LIN {X 0,Y 190.202,Z 1213.13,A -85,B 0,C 180,E1 7235.052,E2 7235.052} C_VEL
LIN {X 0,Y 181.656,Z 1215.666,A -85,B 0,C 180,E1 7232.27,E2 7232.27} C_VEL
LIN {X 0,Y 170.699,Z 1218.765,A -85,B 0,C 180,E1 7227.565,E2 7227.565} C_VEL
LIN {X 0,Y 162.904,Z 1221.055,A -85,B 0,C 180,E1 7223.131,E2 7223.131} C_VEL
LIN {X 0,Y 156.495,Z 1223.066,A -85,B 0,C 180,E1 7218.245,E2 7218.245} C_VEL
LIN {X 0,Y 151.281,Z 1224.964,A -85,B 0,C 180,E1 7212.599,E2 7212.599} C_VEL
LIN {X 0,Y 147.668,Z 1226.836,A -85,B 0,C 180,E1 7206.611,E2 7206.611} C_VEL
LIN {X 0,Y 145.616,Z 1229.303,A -85,B 0,C 180,E1 7198.033,E2 7198.033} C_VEL
LIN {X 0,Y 147.248,Z 1232.369,A -85,B 0,C 180,E1 7187.849,E2 7187.849} C_VEL
LIN {X 0,Y 157.913,Z 1236.155,A -85,B 0,C 180,E1 7174.498,E2 7174.498} C_VEL
LIN {X 0,Y 172.688,Z 1238.099,A -85,B 0,C 180,E1 7165.832,E2 7165.832} C_VEL
LIN {X 0,Y 175.368,Z 1238.372,A -85,B 0,C 180,E1 7164.62,E2 7164.62} C_VEL
LIN {X 0,Y 164.681,Z 1250.11,A -85,B 0,C 180,E1 7159.372,E2 7159.372} C_VEL
LIN {X 0,Y 155.017,Z 1260.363,A -85,B 0,C 180,E1 7153.135,E2 7153.135} C_VEL
LIN {X 0,Y 147.162,Z 1268.783,A -85,B 0,C 180,E1 7146.123,E2 7146.123} C_VEL
LIN {X 0,Y 143.911,Z 1271.432,A -85,B 0,C 180,E1 7143.535,E2 7143.535} C_VEL
LIN {X 0,Y 132.963,Z 1277.212,A -85,B 0,C 180,E1 7136.373,E2 7136.373} C_VEL
LIN {X 0,Y 131.052,Z 1278.703,A -85,B 0,C 180,E1 7133.675,E2 7133.675} C_VEL
LIN {X 0,Y 128.932,Z 1282.473,A -85,B 0,C 180,E1 7124.83,E2 7124.83} C_VEL
LIN {X 0,Y 128.699,Z 1284.323,A -85,B 0,C 180,E1 7117.143,E2 7117.143} C_VEL
LIN {X 0,Y 128.951,Z 1284.94,A -85,B 0,C 180,E1 7110.891,E2 7110.891} C_VEL
LIN {X 0,Y 128.784,Z 1284.684,A -85,B 0,C 180,E1 7105.103,E2 7105.103} C_VEL
LIN {X 0,Y 128.69,Z 1283.094,A -85,B 0,C 180,E1 7097.437,E2 7097.437} C_VEL
LIN {X 0,Y 130.24,Z 1279.703,A -85,B 0,C 180,E1 7088.379,E2 7088.379} C_VEL
LIN {X 0,Y 134.227,Z 1274.587,A -85,B 0,C 180,E1 7079.569,E2 7079.569} C_VEL
LIN {X 0,Y 141.174,Z 1267.225,A -85,B 0,C 180,E1 7070.927,E2 7070.927} C_VEL
LIN {X 0,Y 150.261,Z 1258.18,A -85,B 0,C 180,E1 7063.509,E2 7063.509} C_VEL
LIN {X 0,Y 160.858,Z 1247.554,A -85,B 0,C 180,E1 7057.289,E2 7057.289} C_VEL
LIN {X 0,Y 171.789,Z 1236.049,A -85,B 0,C 180,E1 7052.375,E2 7052.375} C_VEL
LIN {X 0,Y 183.624,Z 1222.614,A -85,B 0,C 180,E1 7048.105,E2 7048.105} C_VEL
LIN {X 0,Y 195.661,Z 1207.553,A -85,B 0,C 180,E1 7044.553,E2 7044.553} C_VEL
LIN {X 0,Y 206.741,Z 1192.05,A -85,B 0,C 180,E1 7041.792,E2 7041.792} C_VEL
LIN {X 0,Y 217.435,Z 1175.098,A -85,B 0,C 180,E1 7039.498,E2 7039.498} C_VEL
LIN {X 0,Y 227.58,Z 1156.363,A -85,B 0,C 180,E1 7037.57,E2 7037.57} C_VEL
LIN {X 0,Y 236.655,Z 1136.35,A -85,B 0,C 180,E1 7036.022,E2 7036.022} C_VEL
LIN {X 0,Y 244.117,Z 1116.061,A -85,B 0,C 180,E1 7034.852,E2 7034.852} C_VEL
LIN {X 0,Y 249.756,Z 1096.487,A -85,B 0,C 180,E1 7034.032,E2 7034.032} C_VEL
LIN {X 0,Y 254.152,Z 1075.647,A -85,B 0,C 180,E1 7033.393,E2 7033.393} C_VEL
LIN {X 0,Y 257.474,Z 1050.007,A -85,B 0,C 180,E1 7032.818,E2 7032.818} C_VEL
LIN {X 0,Y 260.557,Z 1021.82,A -85,B 0,C 180,E1 7032.373,E2 7032.373} C_VEL
LIN {X 0,Y 264.495,Z 989.715,A -85,B 0,C 180,E1 7032.277,E2 7032.277} C_VEL
LIN {X 0,Y 264.76,Z 957.802,A -85,B 0,C 180,E1 7027.95,E2 7027.95} C_VEL
LIN {X 0,Y 266.442,Z 929.886,A -85,B 0,C 180,E1 7024.735,E2 7024.735} C_VEL
LIN {X 0,Y 266.944,Z 923.717,A -85,B 0,C 180,E1 7024.08,E2 7024.08} C_VEL
LIN {X 0,Y 267.411,Z 913.202,A -85,B 0,C 180,E1 7019.41,E2 7019.41} C_VEL
LIN {X 0,Y 268.624,Z 906.957,A -85,B 0,C 180,E1 7016.265,E2 7016.265} C_VEL
LIN {X 0,Y 271.7,Z 898.866,A -85,B 0,C 180,E1 7011.748,E2 7011.748} C_VEL
LIN {X 0,Y 277.101,Z 891.459,A -85,B 0,C 180,E1 7006.648,E2 7006.648} C_VEL
LIN {X 0,Y 277.44,Z 891.39,A -85,B 0,C 180,E1 7006.354,E2 7006.354} C_VEL
LIN {X 0,Y 259.966,Z 1057.824,A -85,B 0,C 180,E1 7003.172,E2 7003.172} C_VEL
LIN {X 0,Y 256.354,Z 1078.331,A -85,B 0,C 180,E1 7002.543,E2 7002.543} C_VEL
LIN {X 0,Y 251.132,Z 1098.893,A -85,B 0,C 180,E1 7001.667,E2 7001.667} C_VEL
LIN {X 0,Y 244.438,Z 1118.855,A -85,B 0,C 180,E1 7000.531,E2 7000.531} C_VEL
LIN {X 0,Y 236.901,Z 1136.955,A -85,B 0,C 180,E1 6999.202,E2 6999.202} C_VEL
LIN {X 0,Y 228.237,Z 1154.356,A -85,B 0,C 180,E1 6997.566,E2 6997.566} C_VEL
LIN {X 0,Y 218.015,Z 1171.667,A -85,B 0,C 180,E1 6995.468,E2 6995.468} C_VEL
LIN {X 0,Y 207.123,Z 1187.56,A -85,B 0,C 180,E1 6992.952,E2 6992.952} C_VEL
LIN {X 0,Y 195.887,Z 1201.926,A -85,B 0,C 180,E1 6989.985,E2 6989.985} C_VEL
LIN {X 0,Y 183.923,Z 1215.491,A -85,B 0,C 180,E1 6986.276,E2 6986.276} C_VEL
LIN {X 0,Y 171.894,Z 1227.707,A -85,B 0,C 180,E1 6981.741,E2 6981.741} C_VEL
LIN {X 0,Y 160.986,Z 1237.804,A -85,B 0,C 180,E1 6976.605,E2 6976.605} C_VEL
LIN {X 0,Y 150.926,Z 1246.477,A -85,B 0,C 180,E1 6970.481,E2 6970.481} C_VEL
LIN {X 0,Y 142.092,Z 1253.744,A -85,B 0,C 180,E1 6963.135,E2 6963.135} C_VEL
LIN {X 0,Y 135.409,Z 1259.191,A -85,B 0,C 180,E1 6954.888,E2 6954.888} C_VEL
LIN {X 0,Y 131.267,Z 1262.741,A -85,B 0,C 180,E1 6946.31,E2 6946.31} C_VEL
LIN {X 0,Y 129.3,Z 1264.71,A -85,B 0,C 180,E1 6937.552,E2 6937.552} C_VEL
LIN {X 0,Y 128.89,Z 1265.289,A -85,B 0,C 180,E1 6929.554,E2 6929.554} C_VEL
LIN {X 0,Y 129.406,Z 1264.614,A -85,B 0,C 180,E1 6921.556,E2 6921.556} C_VEL
LIN {X 0,Y 131.568,Z 1262.487,A -85,B 0,C 180,E1 6912.758,E2 6912.758} C_VEL
LIN {X 0,Y 135.899,Z 1258.805,A -85,B 0,C 180,E1 6904.271,E2 6904.271} C_VEL
LIN {X 0,Y 142.537,Z 1253.449,A -85,B 0,C 180,E1 6896.345,E2 6896.345} C_VEL
LIN {X 0,Y 151.344,Z 1246.237,A -85,B 0,C 180,E1 6889.151,E2 6889.151} C_VEL
LIN {X 0,Y 161.477,Z 1237.497,A -85,B 0,C 180,E1 6883.057,E2 6883.057} C_VEL
LIN {X 0,Y 172.614,Z 1227.163,A -85,B 0,C 180,E1 6877.88,E2 6877.88} C_VEL
LIN {X 0,Y 180.192,Z 1219.524,A -85,B 0,C 180,E1 6874.858,E2 6874.858} C_VEL
LIN {X 0,Y 166.021,Z 1223.23,A -85,B 0,C 180,E1 6869.198,E2 6869.198} C_VEL
LIN {X 0,Y 157.334,Z 1225.582,A -85,B 0,C 180,E1 6864.399,E2 6864.399} C_VEL
LIN {X 0,Y 150.611,Z 1227.559,A -85,B 0,C 180,E1 6859.387,E2 6859.387} C_VEL
LIN {X 0,Y 145.112,Z 1229.463,A -85,B 0,C 180,E1 6853.549,E2 6853.549} C_VEL
LIN {X 0,Y 141.144,Z 1231.414,A -85,B 0,C 180,E1 6846.918,E2 6846.918} C_VEL
LIN {X 0,Y 139.007,Z 1233.771,A -85,B 0,C 180,E1 6838.352,E2 6838.352} C_VEL
LIN {X 0,Y 140.751,Z 1236.859,A -85,B 0,C 180,E1 6827.279,E2 6827.279} C_VEL
LIN {X 0,Y 151.475,Z 1240.492,A -85,B 0,C 180,E1 6813.753,E2 6813.753} C_VEL
LIN {X 0,Y 166.114,Z 1242.561,A -85,B 0,C 180,E1 6804.947,E2 6804.947} C_VEL
LIN {X 0,Y 155.353,Z 1253.519,A -85,B 0,C 180,E1 6799.418,E2 6799.418} C_VEL
LIN {X 0,Y 145.567,Z 1263.173,A -85,B 0,C 180,E1 6792.698,E2 6792.698} C_VEL
LIN {X 0,Y 137.392,Z 1271.411,A -85,B 0,C 180,E1 6784.588,E2 6784.588} C_VEL
LIN {X 0,Y 131.799,Z 1277.771,A -85,B 0,C 180,E1 6775.478,E2 6775.478} C_VEL
LIN {X 0,Y 131.052,Z 1278.703,A -85,B 0,C 180,E1 6773.675,E2 6773.675} C_VEL
LIN {X 0,Y 129.012,Z 1280.314,A -85,B 0,C 180,E1 6770.444,E2 6770.444} C_VEL
LIN {X 0,Y 123.443,Z 1282.376,A -85,B 0,C 180,E1 6764.399,E2 6764.399} C_VEL
LIN {X 0,Y 120.803,Z 1283.402,A -85,B 0,C 180,E1 6759.575,E2 6759.575} C_VEL
LIN {X 0,Y 120.68,Z 1283.603,A -85,B 0,C 180,E1 6758.252,E2 6758.252} C_VEL
LIN {X 0,Y 120.946,Z 1284.28,A -85,B 0,C 180,E1 6751.897,E2 6751.897} C_VEL
LIN {X 0,Y 120.862,Z 1284.165,A -85,B 0,C 180,E1 6746.207,E2 6746.207} C_VEL
LIN {X 0,Y 120.653,Z 1282.984,A -85,B 0,C 180,E1 6738.53,E2 6738.53} C_VEL
LIN {X 0,Y 121.897,Z 1280.096,A -85,B 0,C 180,E1 6729.349,E2 6729.349} C_VEL
LIN {X 0,Y 125.732,Z 1275.36,A -85,B 0,C 180,E1 6719.937,E2 6719.937} C_VEL
LIN {X 0,Y 132.369,Z 1268.778,A -85,B 0,C 180,E1 6711.078,E2 6711.078} C_VEL
LIN {X 0,Y 141.438,Z 1260.425,A -85,B 0,C 180,E1 6703.273,E2 6703.273} C_VEL
LIN {X 0,Y 151.584,Z 1251.084,A -85,B 0,C 180,E1 6697.052,E2 6697.052} C_VEL
LIN {X 0,Y 163.215,Z 1239.802,A -85,B 0,C 180,E1 6691.627,E2 6691.627} C_VEL
LIN {X 0,Y 176.089,Z 1226.257,A -85,B 0,C 180,E1 6686.945,E2 6686.945} C_VEL
LIN {X 0,Y 188.388,Z 1211.935,A -85,B 0,C 180,E1 6683.342,E2 6683.342} C_VEL
LIN {X 0,Y 199.998,Z 1196.799,A -85,B 0,C 180,E1 6680.484,E2 6680.484} C_VEL
LIN {X 0,Y 211.415,Z 1179.946,A -85,B 0,C 180,E1 6678.089,E2 6678.089} C_VEL
LIN {X 0,Y 221.752,Z 1162.307,A -85,B 0,C 180,E1 6676.184,E2 6676.184} C_VEL
LIN {X 0,Y 230.796,Z 1144.223,A -85,B 0,C 180,E1 6674.688,E2 6674.688} C_VEL
LIN {X 0,Y 238.814,Z 1124.974,A -85,B 0,C 180,E1 6673.476,E2 6673.476} C_VEL
LIN {X 0,Y 245.784,Z 1103.885,A -85,B 0,C 180,E1 6672.498,E2 6672.498} C_VEL
LIN {X 0,Y 250.857,Z 1083.368,A -85,B 0,C 180,E1 6671.837,E2 6671.837} C_VEL
LIN {X 0,Y 254.306,Z 1062.63,A -85,B 0,C 180,E1 6671.335,E2 6671.335} C_VEL
LIN {X 0,Y 258.057,Z 1029.137,A -85,B 0,C 180,E1 6670.725,E2 6670.725} C_VEL
LIN {X 0,Y 261.533,Z 1000.333,A -85,B 0,C 180,E1 6670.585,E2 6670.585} C_VEL
LIN {X 0,Y 262.564,Z 991.884,A -85,B 0,C 180,E1 6670.557,E2 6670.557} C_VEL
LIN {X 0,Y 263.401,Z 960.962,A -85,B 0,C 180,E1 6666.374,E2 6666.374} C_VEL
LIN {X 0,Y 265.477,Z 933.239,A -85,B 0,C 180,E1 6663.184,E2 6663.184} C_VEL
LIN {X 0,Y 265.825,Z 929.431,A -85,B 0,C 180,E1 6662.748,E2 6662.748} C_VEL
LIN {X 0,Y 266.599,Z 920.148,A -85,B 0,C 180,E1 6658.549,E2 6658.549} C_VEL
LIN {X 0,Y 267.913,Z 914.319,A -85,B 0,C 180,E1 6655.612,E2 6655.612} C_VEL
LIN {X 0,Y 271.136,Z 906.412,A -85,B 0,C 180,E1 6651.197,E2 6651.197} C_VEL
LIN {X 0,Y 274.63,Z 901.489,A -85,B 0,C 180,E1 6647.796,E2 6647.796} C_VEL
LIN {X 0,Y 257.755,Z 1058.451,A -85,B 0,C 180,E1 6644.868,E2 6644.868} C_VEL
LIN {X 0,Y 254.091,Z 1078.81,A -85,B 0,C 180,E1 6644.263,E2 6644.263} C_VEL
LIN {X 0,Y 248.777,Z 1099.339,A -85,B 0,C 180,E1 6643.419,E2 6643.419} C_VEL
LIN {X 0,Y 242.324,Z 1118.342,A -85,B 0,C 180,E1 6642.385,E2 6642.385} C_VEL
LIN {X 0,Y 234.585,Z 1136.721,A -85,B 0,C 180,E1 6641.099,E2 6641.099} C_VEL
LIN {X 0,Y 225.303,Z 1154.957,A -85,B 0,C 180,E1 6639.449,E2 6639.449} C_VEL
LIN {X 0,Y 214.745,Z 1172.372,A -85,B 0,C 180,E1 6637.402,E2 6637.402} C_VEL
LIN {X 0,Y 203.594,Z 1188.167,A -85,B 0,C 180,E1 6634.967,E2 6634.967} C_VEL
LIN {X 0,Y 192.257,Z 1202.219,A -85,B 0,C 180,E1 6632.139,E2 6632.139} C_VEL
LIN {X 0,Y 179.753,Z 1215.917,A -85,B 0,C 180,E1 6628.475,E2 6628.475} C_VEL
LIN {X 0,Y 167.682,Z 1227.709,A -85,B 0,C 180,E1 6624.185,E2 6624.185} C_VEL
LIN {X 0,Y 156.15,Z 1237.926,A -85,B 0,C 180,E1 6619.073,E2 6619.073} C_VEL
LIN {X 0,Y 145.392,Z 1246.707,A -85,B 0,C 180,E1 6612.905,E2 6612.905} C_VEL
LIN {X 0,Y 135.524,Z 1254.267,A -85,B 0,C 180,E1 6605.13,E2 6605.13} C_VEL
LIN {X 0,Y 128.135,Z 1259.807,A -85,B 0,C 180,E1 6596.407,E2 6596.407} C_VEL
LIN {X 0,Y 123.524,Z 1263.398,A -85,B 0,C 180,E1 6587.222,E2 6587.222} C_VEL
LIN {X 0,Y 121.375,Z 1265.321,A -85,B 0,C 180,E1 6578.048,E2 6578.048} C_VEL
LIN {X 0,Y 120.913,Z 1265.897,A -85,B 0,C 180,E1 6569.524,E2 6569.524} C_VEL
LIN {X 0,Y 121.428,Z 1265.285,A -85,B 0,C 180,E1 6561.474,E2 6561.474} C_VEL
LIN {X 0,Y 123.734,Z 1263.249,A -85,B 0,C 180,E1 6552.115,E2 6552.115} C_VEL
LIN {X 0,Y 128.379,Z 1259.659,A -85,B 0,C 180,E1 6543.144,E2 6543.144} C_VEL
LIN {X 0,Y 135.879,Z 1254.064,A -85,B 0,C 180,E1 6534.455,E2 6534.455} C_VEL
LIN {X 0,Y 145.32,Z 1246.851,A -85,B 0,C 180,E1 6527.064,E2 6527.064} C_VEL
LIN {X 0,Y 156.068,Z 1238.11,A -85,B 0,C 180,E1 6520.887,E2 6520.887} C_VEL
LIN {X 0,Y 167.599,Z 1227.933,A -85,B 0,C 180,E1 6515.77,E2 6515.77} C_VEL
LIN {X 0,Y 170.462,Z 1225.224,A -85,B 0,C 180,E1 6514.577,E2 6514.577} C_VEL
LIN {X 0,Y 161.394,Z 1227.526,A -85,B 0,C 180,E1 6510.945,E2 6510.945} C_VEL
LIN {X 0,Y 151.744,Z 1229.936,A -85,B 0,C 180,E1 6505.779,E2 6505.779} C_VEL
LIN {X 0,Y 144.303,Z 1231.953,A -85,B 0,C 180,E1 6500.271,E2 6500.271} C_VEL
LIN {X 0,Y 138.839,Z 1233.726,A -85,B 0,C 180,E1 6494.6,E2 6494.6} C_VEL
LIN {X 0,Y 134.442,Z 1235.714,A -85,B 0,C 180,E1 6487.264,E2 6487.264} C_VEL
LIN {X 0,Y 132.226,Z 1237.88,A -85,B 0,C 180,E1 6479.134,E2 6479.134} C_VEL
LIN {X 0,Y 134.348,Z 1241.242,A -85,B 0,C 180,E1 6466.223,E2 6466.223} C_VEL
LIN {X 0,Y 144.965,Z 1244.651,A -85,B 0,C 180,E1 6452.922,E2 6452.922} C_VEL
LIN {X 0,Y 156.864,Z 1246.466,A -85,B 0,C 180,E1 6445.313,E2 6445.313} C_VEL
LIN {X 0,Y 145.451,Z 1257.166,A -85,B 0,C 180,E1 6439.129,E2 6439.129} C_VEL
LIN {X 0,Y 135.469,Z 1266.256,A -85,B 0,C 180,E1 6431.628,E2 6431.628} C_VEL
LIN {X 0,Y 127.915,Z 1273.369,A -85,B 0,C 180,E1 6423.175,E2 6423.175} C_VEL
LIN {X 0,Y 123.054,Z 1278.667,A -85,B 0,C 180,E1 6413.973,E2 6413.973} C_VEL
LIN {X 0,Y 120.89,Z 1282.238,A -85,B 0,C 180,E1 6404.369,E2 6404.369} C_VEL
LIN {X 0,Y 120.68,Z 1283.603,A -85,B 0,C 180,E1 6398.252,E2 6398.252} C_VEL
LIN {X 0,Y 119.983,Z 1284.024,A -85,B 0,C 180,E1 6395.112,E2 6395.112} C_VEL
LIN {X 0,Y 117.334,Z 1284.085,A -85,B 0,C 180,E1 6390.703,E2 6390.703} C_VEL
LIN {X 0,Y 112.819,Z 1283.189,A -85,B 0,C 180,E1 6382.452,E2 6382.452} C_VEL
LIN {X 0,Y 112.656,Z 1282.948,A -85,B 0,C 180,E1 6381.003,E2 6381.003} C_VEL
LIN {X 0,Y 113.382,Z 1280.71,A -85,B 0,C 180,E1 6371.493,E2 6371.493} C_VEL
LIN {X 0,Y 116.735,Z 1276.632,A -85,B 0,C 180,E1 6361.34,E2 6361.34} C_VEL
LIN {X 0,Y 123.038,Z 1270.723,A -85,B 0,C 180,E1 6351.861,E2 6351.861} C_VEL
LIN {X 0,Y 131.738,Z 1263.271,A -85,B 0,C 180,E1 6343.682,E2 6343.682} C_VEL
LIN {X 0,Y 142.904,Z 1253.731,A -85,B 0,C 180,E1 6336.429,E2 6336.429} C_VEL
LIN {X 0,Y 155.441,Z 1242.448,A -85,B 0,C 180,E1 6330.468,E2 6330.468} C_VEL
LIN {X 0,Y 167.861,Z 1230.368,A -85,B 0,C 180,E1 6325.921,E2 6325.921} C_VEL
LIN {X 0,Y 180.393,Z 1216.979,A -85,B 0,C 180,E1 6322.242,E2 6322.242} C_VEL
LIN {X 0,Y 192.962,Z 1201.882,A -85,B 0,C 180,E1 6319.18,E2 6319.18} C_VEL
LIN {X 0,Y 204.652,Z 1185.877,A -85,B 0,C 180,E1 6316.752,E2 6316.752} C_VEL
LIN {X 0,Y 215.164,Z 1169.416,A -85,B 0,C 180,E1 6314.863,E2 6314.863} C_VEL
LIN {X 0,Y 225.436,Z 1150.63,A -85,B 0,C 180,E1 6313.219,E2 6313.219} C_VEL
LIN {X 0,Y 234.059,Z 1131.794,A -85,B 0,C 180,E1 6311.98,E2 6311.98} C_VEL
LIN {X 0,Y 241.172,Z 1112.847,A -85,B 0,C 180,E1 6311.038,E2 6311.038} C_VEL
LIN {X 0,Y 247.139,Z 1092.355,A -85,B 0,C 180,E1 6310.28,E2 6310.28} C_VEL
LIN {X 0,Y 251.5,Z 1071.38,A -85,B 0,C 180,E1 6309.752,E2 6309.752} C_VEL
LIN {X 0,Y 255.221,Z 1041.377,A -85,B 0,C 180,E1 6309.127,E2 6309.127} C_VEL
LIN {X 0,Y 258.899,Z 1010.146,A -85,B 0,C 180,E1 6308.85,E2 6308.85} C_VEL
LIN {X 0,Y 260.874,Z 994.241,A -85,B 0,C 180,E1 6308.846,E2 6308.846} C_VEL
LIN {X 0,Y 262.228,Z 964.344,A -85,B 0,C 180,E1 6304.811,E2 6304.811} C_VEL
LIN {X 0,Y 264.693,Z 936.724,A -85,B 0,C 180,E1 6301.637,E2 6301.637} C_VEL
LIN {X 0,Y 264.825,Z 935.424,A -85,B 0,C 180,E1 6301.46,E2 6301.46} C_VEL
LIN {X 0,Y 265.786,Z 927.403,A -85,B 0,C 180,E1 6297.844,E2 6297.844} C_VEL
LIN {X 0,Y 267.3,Z 921.495,A -85,B 0,C 180,E1 6294.849,E2 6294.849} C_VEL
LIN {X 0,Y 270.693,Z 913.812,A -85,B 0,C 180,E1 6290.539,E2 6290.539} C_VEL
LIN {X 0,Y 271.955,Z 911.978,A -85,B 0,C 180,E1 6289.26,E2 6289.26} C_VEL
LIN {X 0,Y 255.774,Z 1059.073,A -85,B 0,C 180,E1 6286.592,E2 6286.592} C_VEL
LIN {X 0,Y 252.02,Z 1079.476,A -85,B 0,C 180,E1 6286.006,E2 6286.006} C_VEL
LIN {X 0,Y 246.658,Z 1099.786,A -85,B 0,C 180,E1 6285.203,E2 6285.203} C_VEL
LIN {X 0,Y 240.027,Z 1118.932,A -85,B 0,C 180,E1 6284.203,E2 6284.203} C_VEL
LIN {X 0,Y 232.12,Z 1137.311,A -85,B 0,C 180,E1 6282.967,E2 6282.967} C_VEL
LIN {X 0,Y 222.618,Z 1155.557,A -85,B 0,C 180,E1 6281.379,E2 6281.379} C_VEL
LIN {X 0,Y 211.967,Z 1172.705,A -85,B 0,C 180,E1 6279.44,E2 6279.44} C_VEL
LIN {X 0,Y 200.71,Z 1188.268,A -85,B 0,C 180,E1 6277.134,E2 6277.134} C_VEL
LIN {X 0,Y 188.628,Z 1202.829,A -85,B 0,C 180,E1 6274.301,E2 6274.301} C_VEL
LIN {X 0,Y 176.239,Z 1215.97,A -85,B 0,C 180,E1 6270.887,E2 6270.887} C_VEL
LIN {X 0,Y 163.792,Z 1227.711,A -85,B 0,C 180,E1 6266.749,E2 6266.749} C_VEL
LIN {X 0,Y 151.615,Z 1238.053,A -85,B 0,C 180,E1 6261.69,E2 6261.69} C_VEL
LIN {X 0,Y 139.576,Z 1247.324,A -85,B 0,C 180,E1 6255.166,E2 6255.166} C_VEL
LIN {X 0,Y 128.995,Z 1254.885,A -85,B 0,C 180,E1 6247.197,E2 6247.197} C_VEL
LIN {X 0,Y 120.959,Z 1260.423,A -85,B 0,C 180,E1 6238.108,E2 6238.108} C_VEL
LIN {X 0,Y 115.947,Z 1263.95,A -85,B 0,C 180,E1 6228.604,E2 6228.604} C_VEL
LIN {X 0,Y 113.46,Z 1265.932,A -85,B 0,C 180,E1 6218.614,E2 6218.614} C_VEL
LIN {X 0,Y 112.936,Z 1266.506,A -85,B 0,C 180,E1 6209.49,E2 6209.49} C_VEL
LIN {X 0,Y 113.519,Z 1265.896,A -85,B 0,C 180,E1 6200.876,E2 6200.876} C_VEL
LIN {X 0,Y 116.105,Z 1263.862,A -85,B 0,C 180,E1 6190.896,E2 6190.896} C_VEL
LIN {X 0,Y 121.232,Z 1260.274,A -85,B 0,C 180,E1 6181.42,E2 6181.42} C_VEL
LIN {X 0,Y 129.384,Z 1254.679,A -85,B 0,C 180,E1 6172.372,E2 6172.372} C_VEL
LIN {X 0,Y 139.503,Z 1247.466,A -85,B 0,C 180,E1 6164.799,E2 6164.799} C_VEL
LIN {X 0,Y 151.141,Z 1238.537,A -85,B 0,C 180,E1 6158.452,E2 6158.452} C_VEL
LIN {X 0,Y 160.461,Z 1230.744,A -85,B 0,C 180,E1 6154.392,E2 6154.392} C_VEL
LIN {X 0,Y 146.148,Z 1234.113,A -85,B 0,C 180,E1 6147.283,E2 6147.283} C_VEL
LIN {X 0,Y 138.314,Z 1236.08,A -85,B 0,C 180,E1 6141.635,E2 6141.635} C_VEL
LIN {X 0,Y 132.23,Z 1237.894,A -85,B 0,C 180,E1 6135.347,E2 6135.347} C_VEL
LIN {X 0,Y 127.931,Z 1239.677,A -85,B 0,C 180,E1 6128.541,E2 6128.541} C_VEL
LIN {X 0,Y 127.389,Z 1245.148,A -85,B 0,C 180,E1 6105.919,E2 6105.919} C_VEL
LIN {X 0,Y 138.807,Z 1248.623,A -85,B 0,C 180,E1 6091.615,E2 6091.615} C_VEL
LIN {X 0,Y 147.614,Z 1249.997,A -85,B 0,C 180,E1 6085.73,E2 6085.73} C_VEL
LIN {X 0,Y 136.652,Z 1259.419,A -85,B 0,C 180,E1 6079.55,E2 6079.55} C_VEL
LIN {X 0,Y 126.564,Z 1267.915,A -85,B 0,C 180,E1 6071.578,E2 6071.578} C_VEL
LIN {X 0,Y 119.089,Z 1274.509,A -85,B 0,C 180,E1 6062.505,E2 6062.505} C_VEL
LIN {X 0,Y 114.494,Z 1279.328,A -85,B 0,C 180,E1 6052.599,E2 6052.599} C_VEL
LIN {X 0,Y 112.771,Z 1282.27,A -85,B 0,C 180,E1 6042.768,E2 6042.768} C_VEL
LIN {X 0,Y 112.874,Z 1283.557,A -85,B 0,C 180,E1 6034.066,E2 6034.066} C_VEL
LIN {X 0,Y 112.976,Z 1283.693,A -85,B 0,C 180,E1 6028.481,E2 6028.481} C_VEL
LIN {X 0,Y 112.676,Z 1283.078,A -85,B 0,C 180,E1 6021.84,E2 6021.84} C_VEL
LIN {X 0,Y 112.656,Z 1282.948,A -85,B 0,C 180,E1 6021.003,E2 6021.003} C_VEL
LIN {X 0,Y 111.848,Z 1282.253,A -85,B 0,C 180,E1 6017.368,E2 6017.368} C_VEL
LIN {X 0,Y 108.879,Z 1280.562,A -85,B 0,C 180,E1 6011.22,E2 6011.22} C_VEL
LIN {X 0,Y 107.356,Z 1278.465,A -85,B 0,C 180,E1 6005.11,E2 6005.11} C_VEL
LIN {X 0,Y 107.882,Z 1277.509,A -85,B 0,C 180,E1 6002.793,E2 6002.793} C_VEL
LIN {X 0,Y 113.786,Z 1272.358,A -85,B 0,C 180,E1 5992.679,E2 5992.679} C_VEL
LIN {X 0,Y 122.75,Z 1265.313,A -85,B 0,C 180,E1 5983.539,E2 5983.539} C_VEL
LIN {X 0,Y 134.236,Z 1256.268,A -85,B 0,C 180,E1 5975.723,E2 5975.723} C_VEL
LIN {X 0,Y 147.02,Z 1245.643,A -85,B 0,C 180,E1 5969.487,E2 5969.487} C_VEL
LIN {X 0,Y 159.697,Z 1234.225,A -85,B 0,C 180,E1 5964.796,E2 5964.796} C_VEL
LIN {X 0,Y 173.274,Z 1220.719,A -85,B 0,C 180,E1 5960.809,E2 5960.809} C_VEL
LIN {X 0,Y 186.712,Z 1205.672,A -85,B 0,C 180,E1 5957.602,E2 5957.602} C_VEL
LIN {X 0,Y 198.892,Z 1190.171,A -85,B 0,C 180,E1 5955.153,E2 5955.153} C_VEL
LIN {X 0,Y 210.495,Z 1173.246,A -85,B 0,C 180,E1 5953.161,E2 5953.161} C_VEL
LIN {X 0,Y 221.413,Z 1154.531,A -85,B 0,C 180,E1 5951.505,E2 5951.505} C_VEL
LIN {X 0,Y 230.867,Z 1135.077,A -85,B 0,C 180,E1 5950.227,E2 5950.227} C_VEL
LIN {X 0,Y 238.106,Z 1116.839,A -85,B 0,C 180,E1 5949.322,E2 5949.322} C_VEL
LIN {X 0,Y 244.475,Z 1096.695,A -85,B 0,C 180,E1 5948.582,E2 5948.582} C_VEL
LIN {X 0,Y 249.401,Z 1075.427,A -85,B 0,C 180,E1 5948.024,E2 5948.024} C_VEL
LIN {X 0,Y 252.736,Z 1052.771,A -85,B 0,C 180,E1 5947.564,E2 5947.564} C_VEL
LIN {X 0,Y 255.998,Z 1024.42,A -85,B 0,C 180,E1 5947.154,E2 5947.154} C_VEL
LIN {X 0,Y 259.431,Z 996.349,A -85,B 0,C 180,E1 5947.084,E2 5947.084} C_VEL
LIN {X 0,Y 261.25,Z 967.726,A -85,B 0,C 180,E1 5943.236,E2 5943.236} C_VEL
LIN {X 0,Y 263.958,Z 941.446,A -85,B 0,C 180,E1 5940.196,E2 5940.196} C_VEL
LIN {X 0,Y 265.038,Z 934.554,A -85,B 0,C 180,E1 5937.08,E2 5937.08} C_VEL
LIN {X 0,Y 266.664,Z 928.855,A -85,B 0,C 180,E1 5934.189,E2 5934.189} C_VEL
LIN {X 0,Y 269.428,Z 922.737,A -85,B 0,C 180,E1 5930.749,E2 5930.749} C_VEL
LIN {X 0,Y 254.014,Z 1059.801,A -85,B 0,C 180,E1 5928.34,E2 5928.34} C_VEL
LIN {X 0,Y 250.158,Z 1080.27,A -85,B 0,C 180,E1 5927.772,E2 5927.772} C_VEL
LIN {X 0,Y 244.785,Z 1100.223,A -85,B 0,C 180,E1 5927.017,E2 5927.017} C_VEL
LIN {X 0,Y 237.976,Z 1119.52,A -85,B 0,C 180,E1 5926.054,E2 5926.054} C_VEL
LIN {X 0,Y 229.911,Z 1137.894,A -85,B 0,C 180,E1 5924.874,E2 5924.874} C_VEL
LIN {X 0,Y 220.192,Z 1156.158,A -85,B 0,C 180,E1 5923.354,E2 5923.354} C_VEL
LIN {X 0,Y 209.286,Z 1173.309,A -85,B 0,C 180,E1 5921.497,E2 5921.497} C_VEL
LIN {X 0,Y 197.61,Z 1189.026,A -85,B 0,C 180,E1 5919.256,E2 5919.256} C_VEL
LIN {X 0,Y 185.28,Z 1203.44,A -85,B 0,C 180,E1 5916.545,E2 5916.545} C_VEL
LIN {X 0,Y 172.46,Z 1216.583,A -85,B 0,C 180,E1 5913.227,E2 5913.227} C_VEL
LIN {X 0,Y 159.509,Z 1228.325,A -85,B 0,C 180,E1 5909.174,E2 5909.174} C_VEL
LIN {X 0,Y 146.48,Z 1238.859,A -85,B 0,C 180,E1 5904.053,E2 5904.053} C_VEL
LIN {X 0,Y 133.994,Z 1247.942,A -85,B 0,C 180,E1 5897.62,E2 5897.62} C_VEL
LIN {X 0,Y 122.652,Z 1255.502,A -85,B 0,C 180,E1 5889.48,E2 5889.48} C_VEL
LIN {X 0,Y 113.903,Z 1261.04,A -85,B 0,C 180,E1 5880.021,E2 5880.021} C_VEL
LIN {X 0,Y 108.353,Z 1264.565,A -85,B 0,C 180,E1 5869.961,E2 5869.961} C_VEL
LIN {X 0,Y 105.555,Z 1266.543,A -85,B 0,C 180,E1 5859.264,E2 5859.264} C_VEL
LIN {X 0,Y 104.964,Z 1267.126,A -85,B 0,C 180,E1 5849.998,E2 5849.998} C_VEL
LIN {X 0,Y 105.624,Z 1266.506,A -85,B 0,C 180,E1 5840.187,E2 5840.187} C_VEL
LIN {X 0,Y 108.53,Z 1264.476,A -85,B 0,C 180,E1 5829.505,E2 5829.505} C_VEL
LIN {X 0,Y 114.208,Z 1260.889,A -85,B 0,C 180,E1 5819.482,E2 5819.482} C_VEL
LIN {X 0,Y 123.078,Z 1255.295,A -85,B 0,C 180,E1 5810.073,E2 5810.073} C_VEL
LIN {X 0,Y 133.924,Z 1248.081,A -85,B 0,C 180,E1 5802.341,E2 5802.341} C_VEL
LIN {X 0,Y 145.996,Z 1239.336,A -85,B 0,C 180,E1 5796.084,E2 5796.084} C_VEL
LIN {X 0,Y 150.521,Z 1235.752,A -85,B 0,C 180,E1 5794.041,E2 5794.041} C_VEL
LIN {X 0,Y 140.507,Z 1237.992,A -85,B 0,C 180,E1 5788.941,E2 5788.941} C_VEL
LIN {X 0,Y 132.28,Z 1239.961,A -85,B 0,C 180,E1 5783.145,E2 5783.145} C_VEL
LIN {X 0,Y 125.829,Z 1241.779,A -85,B 0,C 180,E1 5776.623,E2 5776.623} C_VEL
LIN {X 0,Y 121.041,Z 1243.62,A -85,B 0,C 180,E1 5769.031,E2 5769.031} C_VEL
LIN {X 0,Y 120.338,Z 1248.872,A -85,B 0,C 180,E1 5745.567,E2 5745.567} C_VEL
LIN {X 0,Y 132.139,Z 1252.287,A -85,B 0,C 180,E1 5730.54,E2 5730.54} C_VEL
LIN {X 0,Y 138.219,Z 1253.33,A -85,B 0,C 180,E1 5726.152,E2 5726.152} C_VEL
LIN {X 0,Y 126.186,Z 1262.857,A -85,B 0,C 180,E1 5718.832,E2 5718.832} C_VEL
LIN {X 0,Y 116.372,Z 1270.482,A -85,B 0,C 180,E1 5710.123,E2 5710.123} C_VEL
LIN {X 0,Y 109.412,Z 1276.277,A -85,B 0,C 180,E1 5700.176,E2 5700.176} C_VEL
LIN {X 0,Y 105.598,Z 1280.297,A -85,B 0,C 180,E1 5689.356,E2 5689.356} C_VEL
LIN {X 0,Y 104.696,Z 1282.395,A -85,B 0,C 180,E1 5679.346,E2 5679.346} C_VEL
LIN {X 0,Y 104.976,Z 1283.061,A -85,B 0,C 180,E1 5672.186,E2 5672.186} C_VEL
LIN {X 0,Y 104.924,Z 1283,A -85,B 0,C 180,E1 5666.725,E2 5666.725} C_VEL
LIN {X 0,Y 104.681,Z 1282.053,A -85,B 0,C 180,E1 5658.432,E2 5658.432} C_VEL
LIN {X 0,Y 106.159,Z 1279.373,A -85,B 0,C 180,E1 5647.871,E2 5647.871} C_VEL
LIN {X 0,Y 107.882,Z 1277.509,A -85,B 0,C 180,E1 5642.793,E2 5642.793} C_VEL
LIN {X 0,Y 108.755,Z 1275.839,A -85,B 0,C 180,E1 5638.81,E2 5638.81} C_VEL
LIN {X 0,Y 109.807,Z 1270.455,A -85,B 0,C 180,E1 5628.008,E2 5628.008} C_VEL
LIN {X 0,Y 111.996,Z 1268.324,A -85,B 0,C 180,E1 5624.94,E2 5624.94} C_VEL
LIN {X 0,Y 123.281,Z 1260.246,A -85,B 0,C 180,E1 5616.302,E2 5616.302} C_VEL
LIN {X 0,Y 136.479,Z 1250.31,A -85,B 0,C 180,E1 5609.335,E2 5609.335} C_VEL
LIN {X 0,Y 150.021,Z 1239.209,A -85,B 0,C 180,E1 5604.071,E2 5604.071} C_VEL
LIN {X 0,Y 163.763,Z 1226.73,A -85,B 0,C 180,E1 5599.912,E2 5599.912} C_VEL
LIN {X 0,Y 177.369,Z 1212.882,A -85,B 0,C 180,E1 5596.607,E2 5596.607} C_VEL
LIN {X 0,Y 190.588,Z 1197.61,A -85,B 0,C 180,E1 5593.949,E2 5593.949} C_VEL
LIN {X 0,Y 202.809,Z 1181.46,A -85,B 0,C 180,E1 5591.879,E2 5591.879} C_VEL
LIN {X 0,Y 214.335,Z 1163.725,A -85,B 0,C 180,E1 5590.174,E2 5590.174} C_VEL
LIN {X 0,Y 224.62,Z 1144.896,A -85,B 0,C 180,E1 5588.822,E2 5588.822} C_VEL
LIN {X 0,Y 233.122,Z 1126.08,A -85,B 0,C 180,E1 5587.806,E2 5587.806} C_VEL
LIN {X 0,Y 240.263,Z 1106.532,A -85,B 0,C 180,E1 5587.022,E2 5587.022} C_VEL
LIN {X 0,Y 246.117,Z 1085.588,A -85,B 0,C 180,E1 5586.433,E2 5586.433} C_VEL
LIN {X 0,Y 250.15,Z 1064.763,A -85,B 0,C 180,E1 5585.984,E2 5585.984} C_VEL
LIN {X 0,Y 254.338,Z 1030.51,A -85,B 0,C 180,E1 5585.426,E2 5585.426} C_VEL
LIN {X 0,Y 257.968,Z 1000.776,A -85,B 0,C 180,E1 5585.342,E2 5585.342} C_VEL
LIN {X 0,Y 258.249,Z 998.307,A -85,B 0,C 180,E1 5585.289,E2 5585.289} C_VEL
LIN {X 0,Y 260.472,Z 971.107,A -85,B 0,C 180,E1 5581.649,E2 5581.649} C_VEL
LIN {X 0,Y 263.247,Z 947.275,A -85,B 0,C 180,E1 5578.857,E2 5578.857} C_VEL
LIN {X 0,Y 264.42,Z 941.386,A -85,B 0,C 180,E1 5576.151,E2 5576.151} C_VEL
LIN {X 0,Y 266.14,Z 936.026,A -85,B 0,C 180,E1 5573.42,E2 5573.42} C_VEL
LIN {X 0,Y 267.027,Z 934.014,A -85,B 0,C 180,E1 5572.256,E2 5572.256} C_VEL
LIN {X 0,Y 252.507,Z 1060.427,A -85,B 0,C 180,E1 5570.112,E2 5570.112} C_VEL
LIN {X 0,Y 248.575,Z 1080.9,A -85,B 0,C 180,E1 5569.568,E2 5569.568} C_VEL
LIN {X 0,Y 243.16,Z 1100.665,A -85,B 0,C 180,E1 5568.856,E2 5568.856} C_VEL
LIN {X 0,Y 236.178,Z 1120.109,A -85,B 0,C 180,E1 5567.936,E2 5567.936} C_VEL
LIN {X 0,Y 227.963,Z 1138.474,A -85,B 0,C 180,E1 5566.816,E2 5566.816} C_VEL
LIN {X 0,Y 218.033,Z 1156.758,A -85,B 0,C 180,E1 5565.371,E2 5565.371} C_VEL
LIN {X 0,Y 206.88,Z 1173.913,A -85,B 0,C 180,E1 5563.603,E2 5563.603} C_VEL
LIN {X 0,Y 195.056,Z 1189.45,A -85,B 0,C 180,E1 5561.493,E2 5561.493} C_VEL
LIN {X 0,Y 182.226,Z 1204.051,A -85,B 0,C 180,E1 5558.867,E2 5558.867} C_VEL
LIN {X 0,Y 168.982,Z 1217.196,A -85,B 0,C 180,E1 5555.669,E2 5555.669} C_VEL
LIN {X 0,Y 155.528,Z 1228.94,A -85,B 0,C 180,E1 5551.728,E2 5551.728} C_VEL
LIN {X 0,Y 142.167,Z 1239.28,A -85,B 0,C 180,E1 5546.813,E2 5546.813} C_VEL
LIN {X 0,Y 128.68,Z 1248.559,A -85,B 0,C 180,E1 5540.283,E2 5540.283} C_VEL
LIN {X 0,Y 116.524,Z 1256.119,A -85,B 0,C 180,E1 5532.009,E2 5532.009} C_VEL
LIN {X 0,Y 106.991,Z 1261.656,A -85,B 0,C 180,E1 5522.184,E2 5522.184} C_VEL
LIN {X 0,Y 100.825,Z 1265.179,A -85,B 0,C 180,E1 5511.523,E2 5511.523} C_VEL
LIN {X 0,Y 97.664,Z 1267.154,A -85,B 0,C 180,E1 5500.02,E2 5500.02} C_VEL
LIN {X 0,Y 96.987,Z 1267.735,A -85,B 0,C 180,E1 5489.997,E2 5489.997} C_VEL
LIN {X 0,Y 97.653,Z 1267.178,A -85,B 0,C 180,E1 5479.973,E2 5479.973} C_VEL
LIN {X 0,Y 100.796,Z 1265.237,A -85,B 0,C 180,E1 5468.465,E2 5468.465} C_VEL
LIN {X 0,Y 106.946,Z 1261.743,A -85,B 0,C 180,E1 5457.796,E2 5457.796} C_VEL
LIN {X 0,Y 116.467,Z 1256.223,A -85,B 0,C 180,E1 5447.959,E2 5447.959} C_VEL
LIN {X 0,Y 127.982,Z 1249.082,A -85,B 0,C 180,E1 5440.035,E2 5440.035} C_VEL
LIN {X 0,Y 140.457,Z 1240.576,A -85,B 0,C 180,E1 5433.79,E2 5433.79} C_VEL
LIN {X 0,Y 126.224,Z 1243.591,A -85,B 0,C 180,E1 5424.825,E2 5424.825} C_VEL
LIN {X 0,Y 114.189,Z 1247.187,A -85,B 0,C 180,E1 5410.087,E2 5410.087} C_VEL
LIN {X 0,Y 113.198,Z 1252.41,A -85,B 0,C 180,E1 5385.159,E2 5385.159} C_VEL
LIN {X 0,Y 125.941,Z 1255.847,A -85,B 0,C 180,E1 5368.934,E2 5368.934} C_VEL
LIN {X 0,Y 128.87,Z 1256.394,A -85,B 0,C 180,E1 5366.653,E2 5366.653} C_VEL
LIN {X 0,Y 116.805,Z 1265.149,A -85,B 0,C 180,E1 5358.879,E2 5358.879} C_VEL
LIN {X 0,Y 106.642,Z 1272.418,A -85,B 0,C 180,E1 5348.919,E2 5348.919} C_VEL
LIN {X 0,Y 99.914,Z 1277.681,A -85,B 0,C 180,E1 5337.411,E2 5337.411} C_VEL
LIN {X 0,Y 97.067,Z 1280.758,A -85,B 0,C 180,E1 5326.151,E2 5326.151} C_VEL
LIN {X 0,Y 96.815,Z 1282.269,A -85,B 0,C 180,E1 5315.93,E2 5315.93} C_VEL
LIN {X 0,Y 97.043,Z 1282.525,A -85,B 0,C 180,E1 5309.412,E2 5309.412} C_VEL
LIN {X 0,Y 96.702,Z 1282.004,A -85,B 0,C 180,E1 5301.68,E2 5301.68} C_VEL
LIN {X 0,Y 97.336,Z 1280.209,A -85,B 0,C 180,E1 5291.434,E2 5291.434} C_VEL
LIN {X 0,Y 101.027,Z 1276.5,A -85,B 0,C 180,E1 5279.689,E2 5279.689} C_VEL
LIN {X 0,Y 108.567,Z 1270.748,A -85,B 0,C 180,E1 5268.467,E2 5268.467} C_VEL
LIN {X 0,Y 111.996,Z 1268.324,A -85,B 0,C 180,E1 5264.94,E2 5264.94} C_VEL
LIN {X 0,Y 114.767,Z 1265.763,A -85,B 0,C 180,E1 5261.524,E2 5261.524} C_VEL
LIN {X 0,Y 120.848,Z 1258.347,A -85,B 0,C 180,E1 5252.288,E2 5252.288} C_VEL
LIN {X 0,Y 124.308,Z 1255.599,A -85,B 0,C 180,E1 5249.941,E2 5249.941} C_VEL
LIN {X 0,Y 137.98,Z 1245.559,A -85,B 0,C 180,E1 5244.075,E2 5244.075} C_VEL
LIN {X 0,Y 152.607,Z 1233.676,A -85,B 0,C 180,E1 5239.364,E2 5239.364} C_VEL
LIN {X 0,Y 167.212,Z 1220.322,A -85,B 0,C 180,E1 5235.703,E2 5235.703} C_VEL
LIN {X 0,Y 181.102,Z 1205.887,A -85,B 0,C 180,E1 5232.879,E2 5232.879} C_VEL
LIN {X 0,Y 193.8,Z 1190.825,A -85,B 0,C 180,E1 5230.703,E2 5230.703} C_VEL
LIN {X 0,Y 206.433,Z 1173.424,A -85,B 0,C 180,E1 5228.868,E2 5228.868} C_VEL
LIN {X 0,Y 217.311,Z 1155.774,A -85,B 0,C 180,E1 5227.475,E2 5227.475} C_VEL
LIN {X 0,Y 226.87,Z 1137.361,A -85,B 0,C 180,E1 5226.386,E2 5226.386} C_VEL
LIN {X 0,Y 235.056,Z 1118.208,A -85,B 0,C 180,E1 5225.532,E2 5225.532} C_VEL
LIN {X 0,Y 241.807,Z 1098.314,A -85,B 0,C 180,E1 5224.883,E2 5224.883} C_VEL
LIN {X 0,Y 247.002,Z 1077.8,A -85,B 0,C 180,E1 5224.397,E2 5224.397} C_VEL
LIN {X 0,Y 250.616,Z 1056.06,A -85,B 0,C 180,E1 5224,E2 5224} C_VEL
LIN {X 0,Y 253.974,Z 1027.79,A -85,B 0,C 180,E1 5223.605,E2 5223.605} C_VEL
LIN {X 0,Y 257.301,Z 1000.542,A -85,B 0,C 180,E1 5223.522,E2 5223.522} C_VEL
LIN {X 0,Y 259.883,Z 974.6,A -85,B 0,C 180,E1 5220.068,E2 5220.068} C_VEL
LIN {X 0,Y 262.667,Z 953.168,A -85,B 0,C 180,E1 5217.545,E2 5217.545} C_VEL
LIN {X 0,Y 264.825,Z 945.192,A -85,B 0,C 180,E1 5213.799,E2 5213.799} C_VEL
LIN {X 0,Y 251.23,Z 1061.152,A -85,B 0,C 180,E1 5211.901,E2 5211.901} C_VEL
LIN {X 0,Y 247.245,Z 1081.499,A -85,B 0,C 180,E1 5211.386,E2 5211.386} C_VEL
LIN {X 0,Y 241.478,Z 1102.06,A -85,B 0,C 180,E1 5210.681,E2 5210.681} C_VEL
LIN {X 0,Y 234.172,Z 1121.802,A -85,B 0,C 180,E1 5209.787,E2 5209.787} C_VEL
LIN {X 0,Y 225.817,Z 1139.935,A -85,B 0,C 180,E1 5208.73,E2 5208.73} C_VEL
LIN {X 0,Y 216.149,Z 1157.359,A -85,B 0,C 180,E1 5207.425,E2 5207.425} C_VEL
LIN {X 0,Y 204.761,Z 1174.518,A -85,B 0,C 180,E1 5205.756,E2 5205.756} C_VEL
LIN {X 0,Y 192.657,Z 1190.058,A -85,B 0,C 180,E1 5203.759,E2 5203.759} C_VEL
LIN {X 0,Y 179.482,Z 1204.661,A -85,B 0,C 180,E1 5201.264,E2 5201.264} C_VEL
LIN {X 0,Y 165.824,Z 1217.809,A -85,B 0,C 180,E1 5198.207,E2 5198.207} C_VEL
LIN {X 0,Y 151.872,Z 1229.555,A -85,B 0,C 180,E1 5194.411,E2 5194.411} C_VEL
LIN {X 0,Y 137.908,Z 1239.896,A -85,B 0,C 180,E1 5189.625,E2 5189.625} C_VEL
LIN {X 0,Y 123.667,Z 1249.176,A -85,B 0,C 180,E1 5183.166,E2 5183.166} C_VEL
LIN {X 0,Y 110.648,Z 1256.737,A -85,B 0,C 180,E1 5174.813,E2 5174.813} C_VEL
LIN {X 0,Y 100.251,Z 1262.272,A -85,B 0,C 180,E1 5164.642,E2 5164.642} C_VEL
LIN {X 0,Y 93.386,Z 1265.794,A -85,B 0,C 180,E1 5153.335,E2 5153.335} C_VEL
LIN {X 0,Y 89.792,Z 1267.765,A -85,B 0,C 180,E1 5140.909,E2 5140.909} C_VEL
LIN {X 0,Y 89.01,Z 1268.344,A -85,B 0,C 180,E1 5129.997,E2 5129.997} C_VEL
LIN {X 0,Y 89.781,Z 1267.789,A -85,B 0,C 180,E1 5119.084,E2 5119.084} C_VEL
LIN {X 0,Y 93.355,Z 1265.85,A -85,B 0,C 180,E1 5106.651,E2 5106.651} C_VEL
LIN {X 0,Y 100.207,Z 1262.358,A -85,B 0,C 180,E1 5095.334,E2 5095.334} C_VEL
LIN {X 0,Y 110.592,Z 1256.839,A -85,B 0,C 180,E1 5085.152,E2 5085.152} C_VEL
LIN {X 0,Y 122.933,Z 1249.697,A -85,B 0,C 180,E1 5077.146,E2 5077.146} C_VEL
LIN {X 0,Y 130.412,Z 1245,A -85,B 0,C 180,E1 5073.375,E2 5073.375} C_VEL
LIN {X 0,Y 113.605,Z 1248.583,A -85,B 0,C 180,E1 5060.614,E2 5060.614} C_VEL
LIN {X 0,Y 103.595,Z 1253.848,A -85,B 0,C 180,E1 5034.463,E2 5034.463} C_VEL
LIN {X 0,Y 117.702,Z 1258.834,A -85,B 0,C 180,E1 5008.791,E2 5008.791} C_VEL
LIN {X 0,Y 119.501,Z 1259.195,A -85,B 0,C 180,E1 5007.237,E2 5007.237} C_VEL
LIN {X 0,Y 107.419,Z 1267.137,A -85,B 0,C 180,E1 4998.937,E2 4998.937} C_VEL
LIN {X 0,Y 97.728,Z 1273.436,A -85,B 0,C 180,E1 4988.619,E2 4988.619} C_VEL
LIN {X 0,Y 91.219,Z 1278.158,A -85,B 0,C 180,E1 4976.001,E2 4976.001} C_VEL
LIN {X 0,Y 88.811,Z 1280.911,A -85,B 0,C 180,E1 4963.015,E2 4963.015} C_VEL
LIN {X 0,Y 88.937,Z 1281.782,A -85,B 0,C 180,E1 4953.871,E2 4953.871} C_VEL
LIN {X 0,Y 89.019,Z 1281.864,A -85,B 0,C 180,E1 4948.072,E2 4948.072} C_VEL
LIN {X 0,Y 88.696,Z 1281.224,A -85,B 0,C 180,E1 4939.612,E2 4939.612} C_VEL
LIN {X 0,Y 90.006,Z 1279.178,A -85,B 0,C 180,E1 4927.812,E2 4927.812} C_VEL
LIN {X 0,Y 95.099,Z 1275.089,A -85,B 0,C 180,E1 4915.09,E2 4915.09} C_VEL
LIN {X 0,Y 103.471,Z 1269.462,A -85,B 0,C 180,E1 4904.355,E2 4904.355} C_VEL
LIN {X 0,Y 115.003,Z 1261.906,A -85,B 0,C 180,E1 4895.194,E2 4895.194} C_VEL
LIN {X 0,Y 124.308,Z 1255.599,A -85,B 0,C 180,E1 4889.941,E2 4889.941} C_VEL
LIN {X 0,Y 128.443,Z 1252.336,A -85,B 0,C 180,E1 4887.352,E2 4887.352} C_VEL
LIN {X 0,Y 137.881,Z 1242.96,A -85,B 0,C 180,E1 4880.225,E2 4880.225} C_VEL
LIN {X 0,Y 141.971,Z 1239.522,A -85,B 0,C 180,E1 4878.591,E2 4878.591} C_VEL
LIN {X 0,Y 157.088,Z 1227.045,A -85,B 0,C 180,E1 4874.661,E2 4874.661} C_VEL
LIN {X 0,Y 171.525,Z 1213.512,A -85,B 0,C 180,E1 4871.684,E2 4871.684} C_VEL
LIN {X 0,Y 185.588,Z 1198.411,A -85,B 0,C 180,E1 4869.301,E2 4869.301} C_VEL
LIN {X 0,Y 199.119,Z 1181.545,A -85,B 0,C 180,E1 4867.387,E2 4867.387} C_VEL
LIN {X 0,Y 211.091,Z 1163.991,A -85,B 0,C 180,E1 4865.921,E2 4865.921} C_VEL
LIN {X 0,Y 221.245,Z 1146.389,A -85,B 0,C 180,E1 4864.819,E2 4864.819} C_VEL
LIN {X 0,Y 230.498,Z 1127.136,A -85,B 0,C 180,E1 4863.91,E2 4863.91} C_VEL
LIN {X 0,Y 238.335,Z 1106.824,A -85,B 0,C 180,E1 4863.21,E2 4863.21} C_VEL
LIN {X 0,Y 244.348,Z 1086.484,A -85,B 0,C 180,E1 4862.723,E2 4862.723} C_VEL
LIN {X 0,Y 248.665,Z 1065.882,A -85,B 0,C 180,E1 4862.333,E2 4862.333} C_VEL
LIN {X 0,Y 253.056,Z 1031.734,A -85,B 0,C 180,E1 4861.828,E2 4861.828} C_VEL
LIN {X 0,Y 256.609,Z 1002.675,A -85,B 0,C 180,E1 4861.736,E2 4861.736} C_VEL
LIN {X 0,Y 259.459,Z 978.325,A -85,B 0,C 180,E1 4858.509,E2 4858.509} C_VEL
LIN {X 0,Y 262.227,Z 959.046,A -85,B 0,C 180,E1 4856.228,E2 4856.228} C_VEL
LIN {X 0,Y 262.718,Z 957.232,A -85,B 0,C 180,E1 4855.346,E2 4855.346} C_VEL
LIN {X 0,Y 250.201,Z 1061.88,A -85,B 0,C 180,E1 4853.707,E2 4853.707} C_VEL
LIN {X 0,Y 246.118,Z 1082.308,A -85,B 0,C 180,E1 4853.217,E2 4853.217} C_VEL
LIN {X 0,Y 240.338,Z 1102.569,A -85,B 0,C 180,E1 4852.563,E2 4852.563} C_VEL
LIN {X 0,Y 232.888,Z 1122.39,A -85,B 0,C 180,E1 4851.722,E2 4851.722} C_VEL
LIN {X 0,Y 224.392,Z 1140.53,A -85,B 0,C 180,E1 4850.733,E2 4850.733} C_VEL
LIN {X 0,Y 214.548,Z 1157.959,A -85,B 0,C 180,E1 4849.513,E2 4849.513} C_VEL
LIN {X 0,Y 202.937,Z 1175.122,A -85,B 0,C 180,E1 4847.951,E2 4847.951} C_VEL
LIN {X 0,Y 190.566,Z 1190.666,A -85,B 0,C 180,E1 4846.078,E2 4846.078} C_VEL
LIN {X 0,Y 177.061,Z 1205.272,A -85,B 0,C 180,E1 4843.731,E2 4843.731} C_VEL
LIN {X 0,Y 163.003,Z 1218.422,A -85,B 0,C 180,E1 4840.839,E2 4840.839} C_VEL
LIN {X 0,Y 148.565,Z 1230.169,A -85,B 0,C 180,E1 4837.219,E2 4837.219} C_VEL
LIN {X 0,Y 134.003,Z 1240.513,A -85,B 0,C 180,E1 4832.608,E2 4832.608} C_VEL
LIN {X 0,Y 118.994,Z 1249.793,A -85,B 0,C 180,E1 4826.285,E2 4826.285} C_VEL
LIN {X 0,Y 105.066,Z 1257.354,A -85,B 0,C 180,E1 4817.923,E2 4817.923} C_VEL
LIN {X 0,Y 93.721,Z 1262.889,A -85,B 0,C 180,E1 4807.449,E2 4807.449} C_VEL
LIN {X 0,Y 86.054,Z 1266.408,A -85,B 0,C 180,E1 4795.458,E2 4795.458} C_VEL
LIN {X 0,Y 81.944,Z 1268.376,A -85,B 0,C 180,E1 4781.968,E2 4781.968} C_VEL
LIN {X 0,Y 81.033,Z 1268.952,A -85,B 0,C 180,E1 4769.997,E2 4769.997} C_VEL
LIN {X 0,Y 81.934,Z 1268.399,A -85,B 0,C 180,E1 4758.024,E2 4758.024} C_VEL
LIN {X 0,Y 86.024,Z 1266.464,A -85,B 0,C 180,E1 4744.526,E2 4744.526} C_VEL
LIN {X 0,Y 93.676,Z 1262.973,A -85,B 0,C 180,E1 4732.523,E2 4732.523} C_VEL
LIN {X 0,Y 105.012,Z 1257.454,A -85,B 0,C 180,E1 4722.037,E2 4722.037} C_VEL
LIN {X 0,Y 118.717,Z 1250.043,A -85,B 0,C 180,E1 4713.772,E2 4713.772} C_VEL
LIN {X 0,Y 120.183,Z 1249.141,A -85,B 0,C 180,E1 4712.91,E2 4712.91} C_VEL
LIN {X 0,Y 100.591,Z 1253.615,A -85,B 0,C 180,E1 4693.217,E2 4693.217} C_VEL
LIN {X 0,Y 99.075,Z 1258.85,A -85,B 0,C 180,E1 4662.984,E2 4662.984} C_VEL
LIN {X 0,Y 110.026,Z 1261.734,A -85,B 0,C 180,E1 4647.851,E2 4647.851} C_VEL
LIN {X 0,Y 97.448,Z 1269.228,A -85,B 0,C 180,E1 4638.508,E2 4638.508} C_VEL
LIN {X 0,Y 87.629,Z 1275.062,A -85,B 0,C 180,E1 4626.397,E2 4626.397} C_VEL
LIN {X 0,Y 82.361,Z 1278.723,A -85,B 0,C 180,E1 4613.62,E2 4613.62} C_VEL
LIN {X 0,Y 80.75,Z 1280.703,A -85,B 0,C 180,E1 4600.707,E2 4600.707} C_VEL
LIN {X 0,Y 81.062,Z 1281.285,A -85,B 0,C 180,E1 4591.417,E2 4591.417} C_VEL
LIN {X 0,Y 80.841,Z 1281.1,A -85,B 0,C 180,E1 4584.325,E2 4584.325} C_VEL
LIN {X 0,Y 81.186,Z 1279.741,A -85,B 0,C 180,E1 4572.071,E2 4572.071} C_VEL
LIN {X 0,Y 85.129,Z 1276.583,A -85,B 0,C 180,E1 4558.097,E2 4558.097} C_VEL
LIN {X 0,Y 93.091,Z 1271.635,A -85,B 0,C 180,E1 4545.726,E2 4545.726} C_VEL
LIN {X 0,Y 104.432,Z 1264.91,A -85,B 0,C 180,E1 4535.534,E2 4535.534} C_VEL
LIN {X 0,Y 118.297,Z 1256.276,A -85,B 0,C 180,E1 4527.449,E2 4527.449} C_VEL
LIN {X 0,Y 133.148,Z 1246.112,A -85,B 0,C 180,E1 4521.39,E2 4521.39} C_VEL
LIN {X 0,Y 141.971,Z 1239.522,A -85,B 0,C 180,E1 4518.591,E2 4518.591} C_VEL
LIN {X 0,Y 146.768,Z 1235.476,A -85,B 0,C 180,E1 4516.778,E2 4516.778} C_VEL
LIN {X 0,Y 157.338,Z 1224.948,A -85,B 0,C 180,E1 4511.678,E2 4511.678} C_VEL
LIN {X 0,Y 162.22,Z 1220.251,A -85,B 0,C 180,E1 4510.325,E2 4510.325} C_VEL
LIN {X 0,Y 176.65,Z 1206.256,A -85,B 0,C 180,E1 4507.908,E2 4507.908} C_VEL
LIN {X 0,Y 190.501,Z 1190.673,A -85,B 0,C 180,E1 4505.969,E2 4505.969} C_VEL
LIN {X 0,Y 203.086,Z 1174.211,A -85,B 0,C 180,E1 4504.48,E2 4504.48} C_VEL
LIN {X 0,Y 214.322,Z 1156.997,A -85,B 0,C 180,E1 4503.311,E2 4503.311} C_VEL
LIN {X 0,Y 224.653,Z 1138.162,A -85,B 0,C 180,E1 4502.362,E2 4502.362} C_VEL
LIN {X 0,Y 233.059,Z 1119.574,A -85,B 0,C 180,E1 4501.66,E2 4501.66} C_VEL
LIN {X 0,Y 240.007,Z 1100.384,A -85,B 0,C 180,E1 4501.13,E2 4501.13} C_VEL
LIN {X 0,Y 245.696,Z 1079.34,A -85,B 0,C 180,E1 4500.703,E2 4500.703} C_VEL
LIN {X 0,Y 249.511,Z 1058.433,A -85,B 0,C 180,E1 4500.374,E2 4500.374} C_VEL
LIN {X 0,Y 253.056,Z 1030.194,A -85,B 0,C 180,E1 4500.009,E2 4500.009} C_VEL
LIN {X 0,Y 256.184,Z 1004.691,A -85,B 0,C 180,E1 4499.93,E2 4499.93} C_VEL
LIN {X 0,Y 259.195,Z 982.282,A -85,B 0,C 180,E1 4496.973,E2 4496.973} C_VEL
LIN {X 0,Y 259.435,Z 980.698,A -85,B 0,C 180,E1 4496.758,E2 4496.758} C_VEL
LIN {X 0,Y 249.392,Z 1062.812,A -85,B 0,C 180,E1 4495.522,E2 4495.522} C_VEL
LIN {X 0,Y 245.245,Z 1083.114,A -85,B 0,C 180,E1 4495.062,E2 4495.062} C_VEL
LIN {X 0,Y 239.358,Z 1103.38,A -85,B 0,C 180,E1 4494.449,E2 4494.449} C_VEL
LIN {X 0,Y 231.653,Z 1123.485,A -85,B 0,C 180,E1 4493.653,E2 4493.653} C_VEL
LIN {X 0,Y 222.765,Z 1142.006,A -85,B 0,C 180,E1 4492.708,E2 4492.708} C_VEL
LIN {X 0,Y 212.761,Z 1159.29,A -85,B 0,C 180,E1 4491.574,E2 4491.574} C_VEL
LIN {X 0,Y 200.946,Z 1176.378,A -85,B 0,C 180,E1 4490.12,E2 4490.12} C_VEL
LIN {X 0,Y 187.867,Z 1192.356,A -85,B 0,C 180,E1 4488.307,E2 4488.307} C_VEL
LIN {X 0,Y 174.066,Z 1206.784,A -85,B 0,C 180,E1 4486.103,E2 4486.103} C_VEL
LIN {X 0,Y 159.648,Z 1219.782,A -85,B 0,C 180,E1 4483.373,E2 4483.373} C_VEL
LIN {X 0,Y 143.909,Z 1232.012,A -85,B 0,C 180,E1 4479.706,E2 4479.706} C_VEL
LIN {X 0,Y 128.847,Z 1242.118,A -85,B 0,C 180,E1 4475.215,E2 4475.215} C_VEL
LIN {X 0,Y 113.948,Z 1250.798,A -85,B 0,C 180,E1 4469.302,E2 4469.302} C_VEL
LIN {X 0,Y 99.827,Z 1257.971,A -85,B 0,C 180,E1 4461.37,E2 4461.37} C_VEL
LIN {X 0,Y 87.448,Z 1263.506,A -85,B 0,C 180,E1 4450.668,E2 4450.668} C_VEL
LIN {X 0,Y 78.863,Z 1267.023,A -85,B 0,C 180,E1 4437.972,E2 4437.972} C_VEL
LIN {X 0,Y 74.129,Z 1268.987,A -85,B 0,C 180,E1 4423.252,E2 4423.252} C_VEL
LIN {X 0,Y 73.056,Z 1269.561,A -85,B 0,C 180,E1 4409.997,E2 4409.997} C_VEL
LIN {X 0,Y 74.119,Z 1269.01,A -85,B 0,C 180,E1 4396.739,E2 4396.739} C_VEL
LIN {X 0,Y 78.832,Z 1267.078,A -85,B 0,C 180,E1 4382.009,E2 4382.009} C_VEL
LIN {X 0,Y 87.403,Z 1263.589,A -85,B 0,C 180,E1 4369.299,E2 4369.299} C_VEL
LIN {X 0,Y 99.776,Z 1258.07,A -85,B 0,C 180,E1 4358.585,E2 4358.585} C_VEL
LIN {X 0,Y 110.047,Z 1252.906,A -85,B 0,C 180,E1 4352.417,E2 4352.417} C_VEL
LIN {X 0,Y 89.242,Z 1258.715,A -85,B 0,C 180,E1 4321.285,E2 4321.285} C_VEL
LIN {X 0,Y 91.685,Z 1261.678,A -85,B 0,C 180,E1 4302.222,E2 4302.222} C_VEL
LIN {X 0,Y 100.688,Z 1263.995,A -85,B 0,C 180,E1 4288.654,E2 4288.654} C_VEL
LIN {X 0,Y 88.044,Z 1270.792,A -85,B 0,C 180,E1 4278.553,E2 4278.553} C_VEL
LIN {X 0,Y 78.567,Z 1275.881,A -85,B 0,C 180,E1 4265.467,E2 4265.467} C_VEL
LIN {X 0,Y 73.596,Z 1279.063,A -85,B 0,C 180,E1 4250.383,E2 4250.383} C_VEL
LIN {X 0,Y 72.846,Z 1280.491,A -85,B 0,C 180,E1 4236.308,E2 4236.308} C_VEL
LIN {X 0,Y 73.098,Z 1280.697,A -85,B 0,C 180,E1 4229.22,E2 4229.22} C_VEL
LIN {X 0,Y 72.731,Z 1280.148,A -85,B 0,C 180,E1 4218.907,E2 4218.907} C_VEL
LIN {X 0,Y 74.586,Z 1278.195,A -85,B 0,C 180,E1 4204.601,E2 4204.601} C_VEL
LIN {X 0,Y 81.076,Z 1274.313,A -85,B 0,C 180,E1 4189.87,E2 4189.87} C_VEL
LIN {X 0,Y 91.962,Z 1268.513,A -85,B 0,C 180,E1 4177.473,E2 4177.473} C_VEL
LIN {X 0,Y 106.246,Z 1260.63,A -85,B 0,C 180,E1 4167.802,E2 4167.802} C_VEL
LIN {X 0,Y 121.94,Z 1251.077,A -85,B 0,C 180,E1 4160.818,E2 4160.818} C_VEL
LIN {X 0,Y 137.8,Z 1240.181,A -85,B 0,C 180,E1 4155.808,E2 4155.808} C_VEL
LIN {X 0,Y 153.363,Z 1227.992,A -85,B 0,C 180,E1 4152.069,E2 4152.069} C_VEL
LIN {X 0,Y 162.22,Z 1220.251,A -85,B 0,C 180,E1 4150.325,E2 4150.325} C_VEL
LIN {X 0,Y 167.12,Z 1215.488,A -85,B 0,C 180,E1 4149.066,E2 4149.066} C_VEL
LIN {X 0,Y 178.198,Z 1203.209,A -85,B 0,C 180,E1 4145.231,E2 4145.231} C_VEL
LIN {X 0,Y 182.988,Z 1197.89,A -85,B 0,C 180,E1 4144.288,E2 4144.288} C_VEL
LIN {X 0,Y 197.186,Z 1180.922,A -85,B 0,C 180,E1 4142.705,E2 4142.705} C_VEL
LIN {X 0,Y 209.538,Z 1163.502,A -85,B 0,C 180,E1 4141.516,E2 4141.516} C_VEL
LIN {X 0,Y 220.475,Z 1145.174,A -85,B 0,C 180,E1 4140.592,E2 4140.592} C_VEL
LIN {X 0,Y 229.962,Z 1125.94,A -85,B 0,C 180,E1 4139.869,E2 4139.869} C_VEL
LIN {X 0,Y 237.977,Z 1105.653,A -85,B 0,C 180,E1 4139.322,E2 4139.322} C_VEL
LIN {X 0,Y 244.127,Z 1085.297,A -85,B 0,C 180,E1 4138.932,E2 4138.932} C_VEL
LIN {X 0,Y 248.594,Z 1064.415,A -85,B 0,C 180,E1 4138.614,E2 4138.614} C_VEL
LIN {X 0,Y 252.864,Z 1032.275,A -85,B 0,C 180,E1 4138.206,E2 4138.206} C_VEL
LIN {X 0,Y 255.946,Z 1007.205,A -85,B 0,C 180,E1 4138.165,E2 4138.165} C_VEL
LIN {X 0,Y 248.743,Z 1064.359,A -85,B 0,C 180,E1 4137.337,E2 4137.337} C_VEL
LIN {X 0,Y 244.387,Z 1084.913,A -85,B 0,C 180,E1 4136.895,E2 4136.895} C_VEL
LIN {X 0,Y 238.449,Z 1104.751,A -85,B 0,C 180,E1 4136.332,E2 4136.332} C_VEL
LIN {X 0,Y 230.642,Z 1124.673,A -85,B 0,C 180,E1 4135.599,E2 4135.599} C_VEL
LIN {X 0,Y 221.406,Z 1143.483,A -85,B 0,C 180,E1 4134.71,E2 4134.71} C_VEL
LIN {X 0,Y 211.253,Z 1160.609,A -85,B 0,C 180,E1 4133.668,E2 4133.668} C_VEL
LIN {X 0,Y 199.249,Z 1177.61,A -85,B 0,C 180,E1 4132.331,E2 4132.331} C_VEL
LIN {X 0,Y 185.461,Z 1194.044,A -85,B 0,C 180,E1 4130.597,E2 4130.597} C_VEL
LIN {X 0,Y 171.379,Z 1208.295,A -85,B 0,C 180,E1 4128.554,E2 4128.554} C_VEL
LIN {X 0,Y 156.618,Z 1221.142,A -85,B 0,C 180,E1 4126.011,E2 4126.011} C_VEL
LIN {X 0,Y 140.719,Z 1233.038,A -85,B 0,C 180,E1 4122.636,E2 4122.636} C_VEL
LIN {X 0,Y 123.979,Z 1243.724,A -85,B 0,C 180,E1 4118.034,E2 4118.034} C_VEL
LIN {X 0,Y 107.674,Z 1252.575,A -85,B 0,C 180,E1 4111.899,E2 4111.899} C_VEL
LIN {X 0,Y 92.889,Z 1259.453,A -85,B 0,C 180,E1 4103.828,E2 4103.828} C_VEL
LIN {X 0,Y 80.368,Z 1264.544,A -85,B 0,C 180,E1 4093.173,E2 4093.173} C_VEL
LIN {X 0,Y 70.745,Z 1268.077,A -85,B 0,C 180,E1 4078.716,E2 4078.716} C_VEL
LIN {X 0,Y 66.056,Z 1269.72,A -85,B 0,C 180,E1 4063.119,E2 4063.119} C_VEL
LIN {X 0,Y 65.083,Z 1270.137,A -85,B 0,C 180,E1 4048.235,E2 4048.235} C_VEL
LIN {X 0,Y 66.692,Z 1269.502,A -85,B 0,C 180,E1 4033.446,E2 4033.446} C_VEL
LIN {X 0,Y 72.61,Z 1267.397,A -85,B 0,C 180,E1 4017.514,E2 4017.514} C_VEL
LIN {X 0,Y 82.599,Z 1263.726,A -85,B 0,C 180,E1 4004.419,E2 4004.419} C_VEL
LIN {X 0,Y 95.65,Z 1258.371,A -85,B 0,C 180,E1 3994.325,E2 3994.325} C_VEL
LIN {X 0,Y 99.843,Z 1256.405,A -85,B 0,C 180,E1 3991.776,E2 3991.776} C_VEL
LIN {X 0,Y 84.224,Z 1264.249,A -85,B 0,C 180,E1 3941.307,E2 3941.307} C_VEL
LIN {X 0,Y 91.157,Z 1266.144,A -85,B 0,C 180,E1 3929.51,E2 3929.51} C_VEL
LIN {X 0,Y 77.523,Z 1272.637,A -85,B 0,C 180,E1 3917.326,E2 3917.326} C_VEL
LIN {X 0,Y 68.471,Z 1276.983,A -85,B 0,C 180,E1 3901.719,E2 3901.719} C_VEL
LIN {X 0,Y 64.963,Z 1279.297,A -85,B 0,C 180,E1 3885.172,E2 3885.172} C_VEL
LIN {X 0,Y 65.05,Z 1280.042,A -85,B 0,C 180,E1 3872.481,E2 3872.481} C_VEL
LIN {X 0,Y 64.99,Z 1280.001,A -85,B 0,C 180,E1 3866.476,E2 3866.476} C_VEL
LIN {X 0,Y 65.046,Z 1279.109,A -85,B 0,C 180,E1 3853.023,E2 3853.023} C_VEL
LIN {X 0,Y 69.325,Z 1276.4,A -85,B 0,C 180,E1 3835.777,E2 3835.777} C_VEL
LIN {X 0,Y 79.027,Z 1271.74,A -85,B 0,C 180,E1 3820.618,E2 3820.618} C_VEL
LIN {X 0,Y 92.019,Z 1265.509,A -85,B 0,C 180,E1 3809.633,E2 3809.633} C_VEL
LIN {X 0,Y 107.448,Z 1257.401,A -85,B 0,C 180,E1 3801.486,E2 3801.486} C_VEL
LIN {X 0,Y 124.462,Z 1247.213,A -85,B 0,C 180,E1 3795.426,E2 3795.426} C_VEL
LIN {X 0,Y 141.605,Z 1235.354,A -85,B 0,C 180,E1 3791.06,E2 3791.06} C_VEL
LIN {X 0,Y 158.45,Z 1221.833,A -85,B 0,C 180,E1 3787.83,E2 3787.83} C_VEL
LIN {X 0,Y 173.769,Z 1207.537,A -85,B 0,C 180,E1 3785.496,E2 3785.496} C_VEL
LIN {X 0,Y 182.988,Z 1197.89,A -85,B 0,C 180,E1 3784.288,E2 3784.288} C_VEL
LIN {X 0,Y 187.708,Z 1192.408,A -85,B 0,C 180,E1 3783.412,E2 3783.412} C_VEL
LIN {X 0,Y 198.383,Z 1178.58,A -85,B 0,C 180,E1 3780.488,E2 3780.488} C_VEL
LIN {X 0,Y 202.784,Z 1172.549,A -85,B 0,C 180,E1 3779.823,E2 3779.823} C_VEL
LIN {X 0,Y 214.453,Z 1155.042,A -85,B 0,C 180,E1 3778.91,E2 3778.91} C_VEL
LIN {X 0,Y 225.076,Z 1135.952,A -85,B 0,C 180,E1 3778.181,E2 3778.181} C_VEL
LIN {X 0,Y 232.023,Z 1121.108,A -85,B 0,C 180,E1 3777.743,E2 3777.743} C_VEL
LIN {X 0,Y 222.779,Z 1140.548,A -85,B 0,C 180,E1 3776.944,E2 3776.944} C_VEL
LIN {X 0,Y 211.988,Z 1158.978,A -85,B 0,C 180,E1 3775.972,E2 3775.972} C_VEL
LIN {X 0,Y 200.467,Z 1175.381,A -85,B 0,C 180,E1 3774.849,E2 3774.849} C_VEL
LIN {X 0,Y 187.69,Z 1190.865,A -85,B 0,C 180,E1 3773.46,E2 3773.46} C_VEL
LIN {X 0,Y 172.822,Z 1206.202,A -85,B 0,C 180,E1 3771.606,E2 3771.606} C_VEL
LIN {X 0,Y 157.679,Z 1219.512,A -85,B 0,C 180,E1 3769.37,E2 3769.37} C_VEL
LIN {X 0,Y 141.886,Z 1231.399,A -85,B 0,C 180,E1 3766.517,E2 3766.517} C_VEL
LIN {X 0,Y 125.609,Z 1241.854,A -85,B 0,C 180,E1 3762.779,E2 3762.779} C_VEL
LIN {X 0,Y 108.28,Z 1251.226,A -85,B 0,C 180,E1 3757.421,E2 3757.421} C_VEL
LIN {X 0,Y 92.14,Z 1258.544,A -85,B 0,C 180,E1 3750.235,E2 3750.235} C_VEL
LIN {X 0,Y 77.848,Z 1264.023,A -85,B 0,C 180,E1 3740.405,E2 3740.405} C_VEL
LIN {X 0,Y 65.984,Z 1267.959,A -85,B 0,C 180,E1 3726.221,E2 3726.221} C_VEL
LIN {X 0,Y 58.851,Z 1270.15,A -85,B 0,C 180,E1 3707.802,E2 3707.802} C_VEL
LIN {X 0,Y 57.11,Z 1270.739,A -85,B 0,C 180,E1 3692.002,E2 3692.002} C_VEL
LIN {X 0,Y 58.116,Z 1270.414,A -85,B 0,C 180,E1 3676.058,E2 3676.058} C_VEL
LIN {X 0,Y 63.372,Z 1268.843,A -85,B 0,C 180,E1 3658.619,E2 3658.619} C_VEL
LIN {X 0,Y 73.427,Z 1265.61,A -85,B 0,C 180,E1 3643.8,E2 3643.8} C_VEL
LIN {X 0,Y 87.007,Z 1260.669,A -85,B 0,C 180,E1 3632.693,E2 3632.693} C_VEL
LIN {X 0,Y 89.605,Z 1259.661,A -85,B 0,C 180,E1 3631.071,E2 3631.071} C_VEL
LIN {X 0,Y 77.015,Z 1266.63,A -85,B 0,C 180,E1 3579.482,E2 3579.482} C_VEL
LIN {X 0,Y 81.685,Z 1267.919,A -85,B 0,C 180,E1 3570.6,E2 3570.6} C_VEL
LIN {X 0,Y 68.507,Z 1273.444,A -85,B 0,C 180,E1 3557.83,E2 3557.83} C_VEL
LIN {X 0,Y 59.619,Z 1277.237,A -85,B 0,C 180,E1 3540.212,E2 3540.212} C_VEL
LIN {X 0,Y 56.803,Z 1279.15,A -85,B 0,C 180,E1 3521.169,E2 3521.169} C_VEL
LIN {X 0,Y 57.158,Z 1279.499,A -85,B 0,C 180,E1 3510.004,E2 3510.004} C_VEL
LIN {X 0,Y 56.778,Z 1279.072,A -85,B 0,C 180,E1 3497.805,E2 3497.805} C_VEL
LIN {X 0,Y 59.81,Z 1277.07,A -85,B 0,C 180,E1 3478.791,E2 3478.791} C_VEL
LIN {X 0,Y 68.488,Z 1273.332,A -85,B 0,C 180,E1 3461.886,E2 3461.886} C_VEL
LIN {X 0,Y 82.139,Z 1267.563,A -85,B 0,C 180,E1 3448.791,E2 3448.791} C_VEL
LIN {X 0,Y 97.875,Z 1260.207,A -85,B 0,C 180,E1 3439.983,E2 3439.983} C_VEL
LIN {X 0,Y 114.348,Z 1251.41,A -85,B 0,C 180,E1 3433.942,E2 3433.942} C_VEL
LIN {X 0,Y 131.77,Z 1240.622,A -85,B 0,C 180,E1 3429.465,E2 3429.465} C_VEL
LIN {X 0,Y 149.018,Z 1228.128,A -85,B 0,C 180,E1 3426.162,E2 3426.162} C_VEL
LIN {X 0,Y 165.324,Z 1214.343,A -85,B 0,C 180,E1 3423.743,E2 3423.743} C_VEL
LIN {X 0,Y 180.075,Z 1199.848,A -85,B 0,C 180,E1 3421.968,E2 3421.968} C_VEL
LIN {X 0,Y 193.977,Z 1183.991,A -85,B 0,C 180,E1 3420.585,E2 3420.585} C_VEL
LIN {X 0,Y 202.784,Z 1172.549,A -85,B 0,C 180,E1 3419.823,E2 3419.823} C_VEL
LIN {X 0,Y 202.863,Z 1172.385,A -85,B 0,C 180,E1 3419.471,E2 3419.471} C_VEL
LIN {X 0,Y 201.868,Z 1173.626,A -85,B 0,C 180,E1 3418.892,E2 3418.892} C_VEL
LIN {X 0,Y 198.414,Z 1178.045,A -85,B 0,C 180,E1 3417.892,E2 3417.892} C_VEL
LIN {X 0,Y 188.144,Z 1190.24,A -85,B 0,C 180,E1 3416.166,E2 3416.166} C_VEL
LIN {X 0,Y 181.818,Z 1197.004,A -85,B 0,C 180,E1 3415.375,E2 3415.375} C_VEL
LIN {X 0,Y 166.989,Z 1211.286,A -85,B 0,C 180,E1 3413.671,E2 3413.671} C_VEL
LIN {X 0,Y 150.657,Z 1224.61,A -85,B 0,C 180,E1 3411.426,E2 3411.426} C_VEL
LIN {X 0,Y 133.654,Z 1236.313,A -85,B 0,C 180,E1 3408.513,E2 3408.513} C_VEL
LIN {X 0,Y 117.063,Z 1245.947,A -85,B 0,C 180,E1 3404.82,E2 3404.82} C_VEL
LIN {X 0,Y 100.201,Z 1254.196,A -85,B 0,C 180,E1 3399.707,E2 3399.707} C_VEL
LIN {X 0,Y 82.772,Z 1261.261,A -85,B 0,C 180,E1 3391.855,E2 3391.855} C_VEL
LIN {X 0,Y 67.434,Z 1266.36,A -85,B 0,C 180,E1 3380.387,E2 3380.387} C_VEL
LIN {X 0,Y 56.224,Z 1269.521,A -85,B 0,C 180,E1 3364.68,E2 3364.68} C_VEL
LIN {X 0,Y 50.21,Z 1271.064,A -85,B 0,C 180,E1 3344.998,E2 3344.998} C_VEL
LIN {X 0,Y 49.163,Z 1271.334,A -85,B 0,C 180,E1 3326.497,E2 3326.497} C_VEL
LIN {X 0,Y 51.797,Z 1270.666,A -85,B 0,C 180,E1 3307.285,E2 3307.285} C_VEL
LIN {X 0,Y 60.18,Z 1268.479,A -85,B 0,C 180,E1 3288.345,E2 3288.345} C_VEL
LIN {X 0,Y 73.648,Z 1264.478,A -85,B 0,C 180,E1 3274.085,E2 3274.085} C_VEL
LIN {X 0,Y 79.329,Z 1262.588,A -85,B 0,C 180,E1 3269.962,E2 3269.962} C_VEL
LIN {X 0,Y 69.498,Z 1268.724,A -85,B 0,C 180,E1 3218.036,E2 3218.036} C_VEL
LIN {X 0,Y 72.296,Z 1269.477,A -85,B 0,C 180,E1 3212.042,E2 3212.042} C_VEL
LIN {X 0,Y 59.166,Z 1274.286,A -85,B 0,C 180,E1 3198.043,E2 3198.043} C_VEL
LIN {X 0,Y 50.779,Z 1277.4,A -85,B 0,C 180,E1 3178.206,E2 3178.206} C_VEL
LIN {X 0,Y 48.832,Z 1278.676,A -85,B 0,C 180,E1 3158.246,E2 3158.246} C_VEL
LIN {X 0,Y 49.126,Z 1278.867,A -85,B 0,C 180,E1 3148.839,E2 3148.839} C_VEL
LIN {X 0,Y 49.19,Z 1278.115,A -85,B 0,C 180,E1 3131.026,E2 3131.026} C_VEL
LIN {X 0,Y 54.542,Z 1275.854,A -85,B 0,C 180,E1 3110.094,E2 3110.094} C_VEL
LIN {X 0,Y 66.533,Z 1271.555,A -85,B 0,C 180,E1 3092.702,E2 3092.702} C_VEL
LIN {X 0,Y 82.511,Z 1265.301,A -85,B 0,C 180,E1 3081.089,E2 3081.089} C_VEL
LIN {X 0,Y 99.801,Z 1257.436,A -85,B 0,C 180,E1 3073.652,E2 3073.652} C_VEL
LIN {X 0,Y 117.312,Z 1248.093,A -85,B 0,C 180,E1 3068.648,E2 3068.648} C_VEL
LIN {X 0,Y 134.671,Z 1237.257,A -85,B 0,C 180,E1 3065.11,E2 3065.11} C_VEL
LIN {X 0,Y 151.127,Z 1225.306,A -85,B 0,C 180,E1 3062.585,E2 3062.585} C_VEL
LIN {X 0,Y 166.982,Z 1211.942,A -85,B 0,C 180,E1 3060.657,E2 3060.657} C_VEL
LIN {X 0,Y 182.49,Z 1196.649,A -85,B 0,C 180,E1 3059.117,E2 3059.117} C_VEL
LIN {X 0,Y 196.681,Z 1180.187,A -85,B 0,C 180,E1 3057.96,E2 3057.96} C_VEL
LIN {X 0,Y 203.573,Z 1171.136,A -85,B 0,C 180,E1 3057.466,E2 3057.466} C_VEL
LIN {X 0,Y 190.376,Z 1187.683,A -85,B 0,C 180,E1 3056.246,E2 3056.246} C_VEL
LIN {X 0,Y 181.818,Z 1197.004,A -85,B 0,C 180,E1 3055.375,E2 3055.375} C_VEL
LIN {X 0,Y 176.337,Z 1202.566,A -85,B 0,C 180,E1 3055.115,E2 3055.115} C_VEL
LIN {X 0,Y 161.469,Z 1215.974,A -85,B 0,C 180,E1 3055.542,E2 3055.542} C_VEL
LIN {X 0,Y 155.469,Z 1220.773,A -85,B 0,C 180,E1 3055.208,E2 3055.208} C_VEL
LIN {X 0,Y 138.764,Z 1232.786,A -85,B 0,C 180,E1 3052.963,E2 3052.963} C_VEL
LIN {X 0,Y 121.807,Z 1243.086,A -85,B 0,C 180,E1 3050.058,E2 3050.058} C_VEL
LIN {X 0,Y 103.156,Z 1252.46,A -85,B 0,C 180,E1 3045.747,E2 3045.747} C_VEL
LIN {X 0,Y 85.273,Z 1259.779,A -85,B 0,C 180,E1 3039.714,E2 3039.714} C_VEL
LIN {X 0,Y 68.686,Z 1265.257,A -85,B 0,C 180,E1 3030.851,E2 3030.851} C_VEL
LIN {X 0,Y 53.827,Z 1269.19,A -85,B 0,C 180,E1 3016.415,E2 3016.415} C_VEL
LIN {X 0,Y 43.861,Z 1271.374,A -85,B 0,C 180,E1 2994.219,E2 2994.219} C_VEL
LIN {X 0,Y 41.167,Z 1271.957,A -85,B 0,C 180,E1 2972.778,E2 2972.778} C_VEL
LIN {X 0,Y 42.749,Z 1271.636,A -85,B 0,C 180,E1 2950.88,E2 2950.88} C_VEL
LIN {X 0,Y 50.347,Z 1270.067,A -85,B 0,C 180,E1 2929,E2 2929} C_VEL
LIN {X 0,Y 63.326,Z 1266.841,A -85,B 0,C 180,E1 2913.188,E2 2913.188} C_VEL
LIN {X 0,Y 68.936,Z 1265.245,A -85,B 0,C 180,E1 2908.859,E2 2908.859} C_VEL
LIN {X 0,Y 62.929,Z 1270.866,A -85,B 0,C 180,E1 2853.867,E2 2853.867} C_VEL
LIN {X 0,Y 48.603,Z 1275.273,A -85,B 0,C 180,E1 2836.063,E2 2836.063} C_VEL
LIN {X 0,Y 41.609,Z 1277.512,A -85,B 0,C 180,E1 2812.618,E2 2812.618} C_VEL
LIN {X 0,Y 41.129,Z 1278.262,A -85,B 0,C 180,E1 2791.399,E2 2791.399} C_VEL
LIN {X 0,Y 40.801,Z 1278.051,A -85,B 0,C 180,E1 2780.129,E2 2780.129} C_VEL
LIN {X 0,Y 44.351,Z 1276.474,A -85,B 0,C 180,E1 2754.123,E2 2754.123} C_VEL
LIN {X 0,Y 55.193,Z 1273.199,A -85,B 0,C 180,E1 2733.567,E2 2733.567} C_VEL
LIN {X 0,Y 71.276,Z 1267.898,A -85,B 0,C 180,E1 2719.981,E2 2719.981} C_VEL
LIN {X 0,Y 89.796,Z 1260.593,A -85,B 0,C 180,E1 2711.533,E2 2711.533} C_VEL
LIN {X 0,Y 108.618,Z 1251.644,A -85,B 0,C 180,E1 2706.216,E2 2706.216} C_VEL
LIN {X 0,Y 126.825,Z 1241.324,A -85,B 0,C 180,E1 2702.71,E2 2702.71} C_VEL
LIN {X 0,Y 143.976,Z 1229.874,A -85,B 0,C 180,E1 2700.255,E2 2700.255} C_VEL
LIN {X 0,Y 161.037,Z 1216.537,A -85,B 0,C 180,E1 2698.374,E2 2698.374} C_VEL
LIN {X 0,Y 173.804,Z 1205.054,A -85,B 0,C 180,E1 2697.192,E2 2697.192} C_VEL
LIN {X 0,Y 158.449,Z 1218.471,A -85,B 0,C 180,E1 2695.555,E2 2695.555} C_VEL
LIN {X 0,Y 155.469,Z 1220.773,A -85,B 0,C 180,E1 2695.208,E2 2695.208} C_VEL
LIN {X 0,Y 149.302,Z 1225.503,A -85,B 0,C 180,E1 2694.834,E2 2694.834} C_VEL
LIN {X 0,Y 132.668,Z 1236.739,A -85,B 0,C 180,E1 2695.164,E2 2695.164} C_VEL
LIN {X 0,Y 126.077,Z 1240.632,A -85,B 0,C 180,E1 2694.68,E2 2694.68} C_VEL
LIN {X 0,Y 108.14,Z 1249.998,A -85,B 0,C 180,E1 2691.599,E2 2691.599} C_VEL
LIN {X 0,Y 90.191,Z 1257.709,A -85,B 0,C 180,E1 2687.295,E2 2687.295} C_VEL
LIN {X 0,Y 71.171,Z 1264.202,A -85,B 0,C 180,E1 2680.252,E2 2680.252} C_VEL
LIN {X 0,Y 53.285,Z 1268.862,A -85,B 0,C 180,E1 2668.302,E2 2668.302} C_VEL
LIN {X 0,Y 39.915,Z 1271.467,A -85,B 0,C 180,E1 2648.765,E2 2648.765} C_VEL
LIN {X 0,Y 33.674,Z 1272.468,A -85,B 0,C 180,E1 2621.988,E2 2621.988} C_VEL
LIN {X 0,Y 33.528,Z 1272.494,A -85,B 0,C 180,E1 2599.685,E2 2599.685} C_VEL
LIN {X 0,Y 39.382,Z 1271.606,A -85,B 0,C 180,E1 2572.451,E2 2572.451} C_VEL
LIN {X 0,Y 53.007,Z 1268.975,A -85,B 0,C 180,E1 2551.884,E2 2551.884} C_VEL
LIN {X 0,Y 58.583,Z 1267.619,A -85,B 0,C 180,E1 2546.948,E2 2546.948} C_VEL
LIN {X 0,Y 53.53,Z 1271.948,A -85,B 0,C 180,E1 2496.252,E2 2496.252} C_VEL
LIN {X 0,Y 39.099,Z 1275.615,A -85,B 0,C 180,E1 2475.736,E2 2475.736} C_VEL
LIN {X 0,Y 32.917,Z 1277.402,A -85,B 0,C 180,E1 2444.072,E2 2444.072} C_VEL
LIN {X 0,Y 33.184,Z 1277.669,A -85,B 0,C 180,E1 2430.008,E2 2430.008} C_VEL
LIN {X 0,Y 34.122,Z 1276.865,A -85,B 0,C 180,E1 2402.049,E2 2402.049} C_VEL
LIN {X 0,Y 43.159,Z 1274.589,A -85,B 0,C 180,E1 2375.832,E2 2375.832} C_VEL
LIN {X 0,Y 59.209,Z 1270.282,A -85,B 0,C 180,E1 2358.988,E2 2358.988} C_VEL
LIN {X 0,Y 78.067,Z 1264.023,A -85,B 0,C 180,E1 2349.552,E2 2349.552} C_VEL
LIN {X 0,Y 97.221,Z 1256.16,A -85,B 0,C 180,E1 2344.027,E2 2344.027} C_VEL
LIN {X 0,Y 115.982,Z 1246.82,A -85,B 0,C 180,E1 2340.464,E2 2340.464} C_VEL
LIN {X 0,Y 134.056,Z 1236.093,A -85,B 0,C 180,E1 2338.022,E2 2338.022} C_VEL
LIN {X 0,Y 143.676,Z 1229.594,A -85,B 0,C 180,E1 2336.965,E2 2336.965} C_VEL
LIN {X 0,Y 126.077,Z 1240.632,A -85,B 0,C 180,E1 2334.68,E2 2334.68} C_VEL
LIN {X 0,Y 119.353,Z 1244.41,A -85,B 0,C 180,E1 2334.127,E2 2334.127} C_VEL
LIN {X 0,Y 101.284,Z 1253.267,A -85,B 0,C 180,E1 2334.301,E2 2334.301} C_VEL
LIN {X 0,Y 94.229,Z 1256.182,A -85,B 0,C 180,E1 2333.564,E2 2333.564} C_VEL
LIN {X 0,Y 74.467,Z 1263.113,A -85,B 0,C 180,E1 2328.55,E2 2328.55} C_VEL
LIN {X 0,Y 55.268,Z 1268.203,A -85,B 0,C 180,E1 2320.161,E2 2320.161} C_VEL
LIN {X 0,Y 38.874,Z 1271.365,A -85,B 0,C 180,E1 2305.379,E2 2305.379} C_VEL
LIN {X 0,Y 27.344,Z 1272.959,A -85,B 0,C 180,E1 2276.016,E2 2276.016} C_VEL
LIN {X 0,Y 25.31,Z 1273.161,A -85,B 0,C 180,E1 2243.184,E2 2243.184} C_VEL
LIN {X 0,Y 30.469,Z 1272.561,A -85,B 0,C 180,E1 2211.418,E2 2211.418} C_VEL
LIN {X 0,Y 44.261,Z 1270.47,A -85,B 0,C 180,E1 2188.223,E2 2188.223} C_VEL
LIN {X 0,Y 48.192,Z 1269.77,A -85,B 0,C 180,E1 2184.519,E2 2184.519} C_VEL
LIN {X 0,Y 44.042,Z 1272.885,A -85,B 0,C 180,E1 2139.484,E2 2139.484} C_VEL
LIN {X 0,Y 29.571,Z 1275.831,A -85,B 0,C 180,E1 2115.252,E2 2115.252} C_VEL
LIN {X 0,Y 24.876,Z 1276.93,A -85,B 0,C 180,E1 2079.262,E2 2079.262} C_VEL
LIN {X 0,Y 25.038,Z 1277.027,A -85,B 0,C 180,E1 2067.721,E2 2067.721} C_VEL
LIN {X 0,Y 27.998,Z 1276.065,A -85,B 0,C 180,E1 2030.009,E2 2030.009} C_VEL
LIN {X 0,Y 42.097,Z 1273.235,A -85,B 0,C 180,E1 2002.15,E2 2002.15} C_VEL
LIN {X 0,Y 60.772,Z 1268.555,A -85,B 0,C 180,E1 1989.222,E2 1989.222} C_VEL
LIN {X 0,Y 80.068,Z 1262.316,A -85,B 0,C 180,E1 1982.627,E2 1982.627} C_VEL
LIN {X 0,Y 100.012,Z 1254.209,A -85,B 0,C 180,E1 1978.581,E2 1978.581} C_VEL
LIN {X 0,Y 112.791,Z 1247.981,A -85,B 0,C 180,E1 1976.702,E2 1976.702} C_VEL
LIN {X 0,Y 94.229,Z 1256.182,A -85,B 0,C 180,E1 1973.564,E2 1973.564} C_VEL
LIN {X 0,Y 87.086,Z 1258.952,A -85,B 0,C 180,E1 1972.704,E2 1972.704} C_VEL
LIN {X 0,Y 67.412,Z 1265.407,A -85,B 0,C 180,E1 1972.527,E2 1972.527} C_VEL
LIN {X 0,Y 60.577,Z 1267.136,A -85,B 0,C 180,E1 1971.241,E2 1971.241} C_VEL
LIN {X 0,Y 41.073,Z 1271.037,A -85,B 0,C 180,E1 1961.673,E2 1961.673} C_VEL
LIN {X 0,Y 24.032,Z 1273.212,A -85,B 0,C 180,E1 1938.478,E2 1938.478} C_VEL
LIN {X 0,Y 17.298,Z 1273.784,A -85,B 0,C 180,E1 1896.624,E2 1896.624} C_VEL
LIN {X 0,Y 20.972,Z 1273.53,A -85,B 0,C 180,E1 1851.685,E2 1851.685} C_VEL
LIN {X 0,Y 35.781,Z 1271.914,A -85,B 0,C 180,E1 1822.741,E2 1822.741} C_VEL
LIN {X 0,Y 37.823,Z 1271.625,A -85,B 0,C 180,E1 1820.463,E2 1820.463} C_VEL
LIN {X 0,Y 35.015,Z 1273.579,A -85,B 0,C 180,E1 1784.784,E2 1784.784} C_VEL
LIN {X 0,Y 20.006,Z 1275.807,A -85,B 0,C 180,E1 1754.421,E2 1754.421} C_VEL
LIN {X 0,Y 17.099,Z 1276.442,A -85,B 0,C 180,E1 1710.015,E2 1710.015} C_VEL
LIN {X 0,Y 21.685,Z 1275.524,A -85,B 0,C 180,E1 1658.405,E2 1658.405} C_VEL
LIN {X 0,Y 38.792,Z 1272.781,A -85,B 0,C 180,E1 1631.671,E2 1631.671} C_VEL
LIN {X 0,Y 58.021,Z 1268.47,A -85,B 0,C 180,E1 1621.964,E2 1621.964} C_VEL
LIN {X 0,Y 78.091,Z 1262.417,A -85,B 0,C 180,E1 1617.004,E2 1617.004} C_VEL
LIN {X 0,Y 81.144,Z 1261.295,A -85,B 0,C 180,E1 1616.402,E2 1616.402} C_VEL
LIN {X 0,Y 61.649,Z 1266.87,A -85,B 0,C 180,E1 1611.592,E2 1611.592} C_VEL
LIN {X 0,Y 60.577,Z 1267.136,A -85,B 0,C 180,E1 1611.241,E2 1611.241} C_VEL
LIN {X 0,Y 53.189,Z 1268.869,A -85,B 0,C 180,E1 1609.578,E2 1609.578} C_VEL
LIN {X 0,Y 32.275,Z 1272.604,A -85,B 0,C 180,E1 1607.85,E2 1607.85} C_VEL
LIN {X 0,Y 25.887,Z 1273.316,A -85,B 0,C 180,E1 1604.292,E2 1604.292} C_VEL
LIN {X 0,Y 10.838,Z 1274.316,A -85,B 0,C 180,E1 1563.582,E2 1563.582} C_VEL
LIN {X 0,Y 10.833,Z 1274.323,A -85,B 0,C 180,E1 1496.346,E2 1496.346} C_VEL
LIN {X 0,Y 25.687,Z 1273.372,A -85,B 0,C 180,E1 1455.816,E2 1455.816} C_VEL
LIN {X 0,Y 27.964,Z 1273.127,A -85,B 0,C 180,E1 1453.549,E2 1453.549} C_VEL
LIN {X 0,Y 26.315,Z 1273.973,A -85,B 0,C 180,E1 1433.46,E2 1433.46} C_VEL
LIN {X 0,Y 9.927,Z 1275.614,A -85,B 0,C 180,E1 1387.214,E2 1387.214} C_VEL
LIN {X 0,Y 8.997,Z 1275.823,A -85,B 0,C 180,E1 1349.349,E2 1349.349} C_VEL
LIN {X 0,Y 18.674,Z 1274.809,A -85,B 0,C 180,E1 1275.521,E2 1275.521} C_VEL
LIN {X 0,Y 38.997,Z 1271.966,A -85,B 0,C 180,E1 1258.894,E2 1258.894} C_VEL
LIN {X 0,Y 47.931,Z 1270.238,A -85,B 0,C 180,E1 1256.002,E2 1256.002} C_VEL
LIN {X 0,Y 28.751,Z 1273.002,A -85,B 0,C 180,E1 1246.797,E2 1246.797} C_VEL
LIN {X 0,Y 25.887,Z 1273.316,A -85,B 0,C 180,E1 1244.292,E2 1244.292} C_VEL
LIN {X 0,Y 20.862,Z 1273.833,A -85,B 0,C 180,E1 1241.287,E2 1241.287} C_VEL
LIN {X 0,Y 5.682,Z 1274.899,A -85,B 0,C 180,E1 1243.377,E2 1243.377} C_VEL
LIN {X 0,Y 2.089,Z 1275.008,A -85,B 0,C 180,E1 1223.923,E2 1223.923} C_VEL
LIN {X 0,Y 8.422,Z 1274.896,A -85,B 0,C 180,E1 1085.425,E2 1085.425} C_VEL
LIN {X 0,Y 0.91,Z 1275.206,A -85,B 0,C 180,E1 990.279,E2 990.279} C_VEL
LIN {X 0,Y 8.044,Z 1274.891,A -85,B 0,C 180,E1 893.616,E2 893.616} C_VEL
LIN {X 0,Y 2.089,Z 1275.008,A -85,B 0,C 180,E1 863.923,E2 863.923} C_VEL
LIN {X 0,Y 1.306,Z 1277.008,A -85,B 0,C 180,E1 798.085,E2 798.085} C_VEL
LIN {X 0,Y 1.306,Z 1319.5,A -85,B 0,C 180,E1 798.085,E2 798.085} C_VEL
LIN {X 0,Y 1.306,Z 1319.5,A -85,B 0,C 180,E1 798.085,E2 798.085}

QRS_NEXT_CUT()

QRS_NEXT()
QRS_HOME()

END
